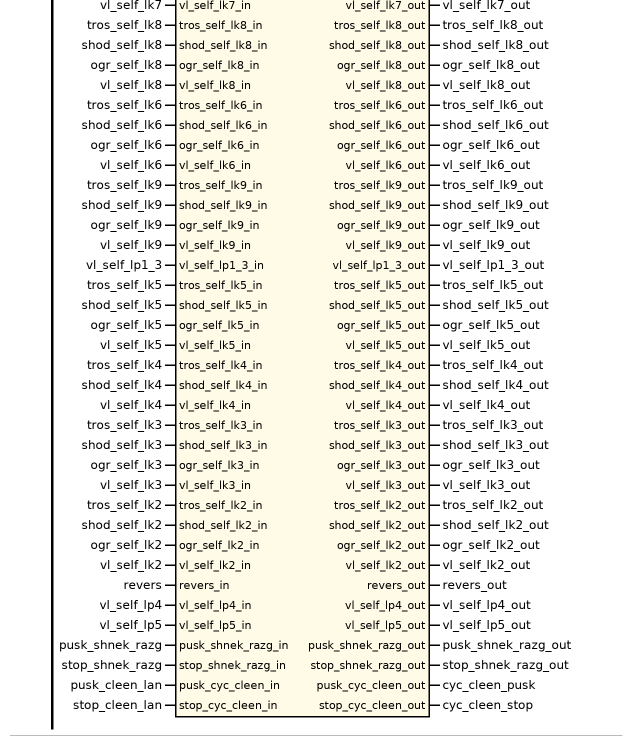
[picture p24: PLC_PRG (LD)]
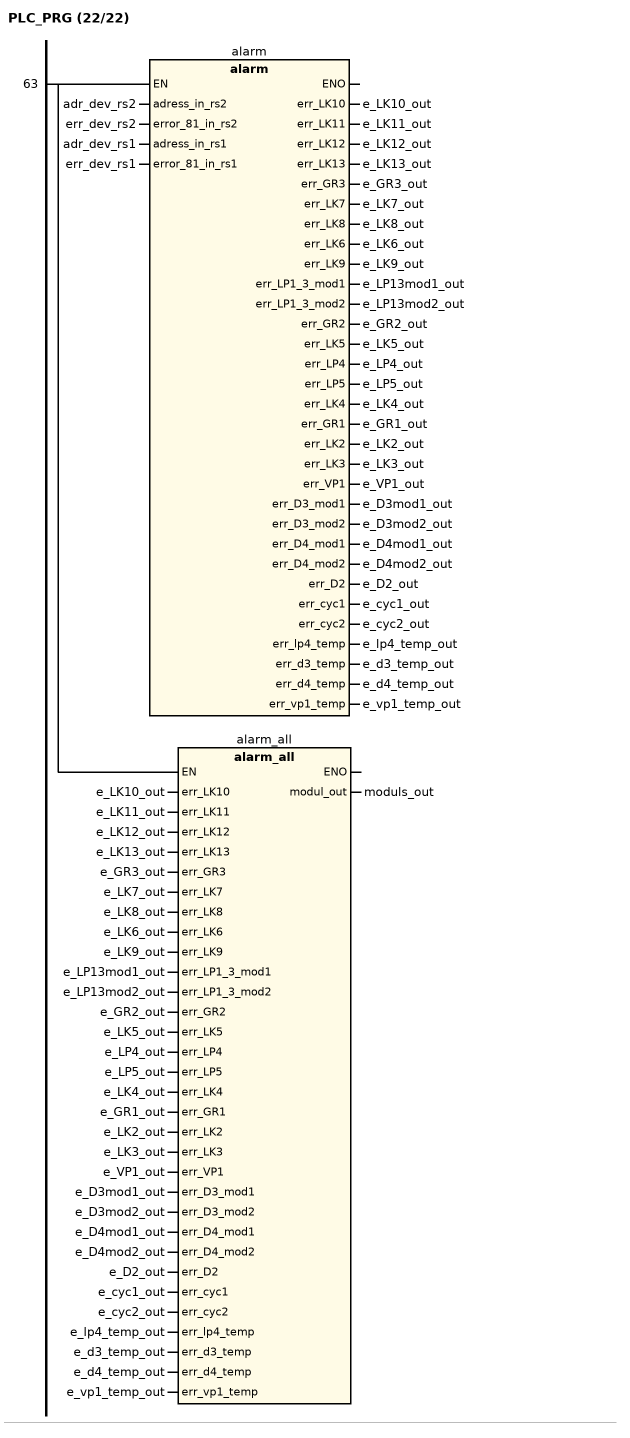
_LD_ (* Ladder Diagram *)
NETWORK 1 (* Фиксация пуска для SCADA-системы *)
	{ [pusk_sys] - [avto_all] | [pusk_lan] } - [/stop_DDD] - [/gribok] --- (pusk_lan)
NETWORK 2 (* Пуск только по готовностям всех шкафов *)
	[pusk_sys] - [avto_all] - [ready_D2] - [ready_D3] - { [ready_D4] | [in_040] } - [ready_LK10] - [ready_LK11] - { [ready_LK12] | [/current_value_lk_glob] } - [ready_LK13] - [ready_GR3] - { [ready_LK7] | [in_040] } - [ready_LK8] - [ready_LK9] - { [ready_LK6] | [in_020] } - [ready_LP1_3] - [ready_GR2] - [ready_LK5] - [ready_LP4] - { [ready_LP5] | [in_040] } - [ready_GR1] - [ready_LK2] - [ready_VP1] - [ready_LK3] --- (pusk)
NETWORK 3 (* Остановка всех агрегатов по втором нажатии кнопки "стоп" *)
	[stop_sys] - stop:CTU(CU: *, RESET: stop_DDD OR pusk_sys OR ruchnoe_all, PV: 2) --- (stop_all)
NETWORK 4 (* Остановка дробилок по третьему нажатию кнопки "стоп" *)
	[stop_sys] - stop_Drob:CTU(CU: *, RESET: stop_DDD OR pusk_sys, PV: 3) --- (stop_D2)
NETWORK 5
	*
		EN --- cyclone:cyclone(stop: stop_DDD, grib: gribok, pusk_LAN: pusk_lan_cyclone_out, stop_lan: stop_lan_cyclone_out, level: lev_up_cyc, KU: ku_cyc, TZ: tz_cyc, skvaj: skvaj_in, switch: revers_out, err: e_cyc1_out OR e_cyc2_out, pusk_shnek_lan: pusk_shnek_razg_out, stop_shnek_lan: stop_shnek_razg_out, in_time: in_time_shake, time_run: time_run, time_stop: time_stop, cleen_in_pusk: cyc_cleen_pusk, cleen_in_stop: cyc_cleen_stop, VE_1 => ve1_out, VE_2 => ve2_out, VE_3 => ve3_out, VE_4 => ve4_out, VE_5 => ve5_out, VE_6 => ve6_out, VE_7 => ve7_out, VE_8 => ve8_out, shnek_up => shnek_up_cyc, ready => ready_cyc, work => work_cyc, avar => avar_cyc, shnek_razg => shnek_razg, prom_cleen_word => prom_cleen_out) => vent_pump_cyc
NETWORK 6
	*
		EN --- PACK(shnek_razg, vent_pump_cyc, shnek_up_cyc, FALSE, FALSE, FALSE, FALSE, FALSE) => km_byte_cyc
NETWORK 7 (* Блок управления дробилкой Д2 *)
	[pusk] - D2:D2(pusk: *, KUD2: KU_D2, RMS2_2: RMS2_2, RD2: RD2_D2, TZD2: TZD2, avto: avto_D2, GRIB: gribok, stop_s: stop_D2, ruchnoe: ruchnoe_all, pusk_LAN: pusk_LAN_D2_out, stop_LAN: stop_LAN_D2_out, err: e_D2_out, work => work_D2, KM2 => KM2_D2, KM3 => KM3_D2, stop_D3D4 => stop_D3, avar => avar_D2) --- (ready_D2)
NETWORK 8 (* Блок управления битовой маской выходов модуля расширения в шкафу управления Д2 *)
	*
		EN --- PACK(FALSE, KM2_D2, FALSE, KM3_D2, FALSE, FALSE, FALSE, FALSE) => KM_D2_byte
NETWORK 9 (* Блок управления дробилкой Д3 *)
	[pusk] - D3:D3(pusk: *, KU: KU_D3, TZN: TZN_D3, KPM: KPM_D3, TZV: TZV_D3, KUD3: KUD3_D3, TZD3: TZD3_D3, RD3: RD3_D3, TM: TM_D3, RMS: RMS_D3, avto_in: avto_D3, GRIB: gribok, work_D2_D3: work_D2, stop_in: stop_D2, ruchnoe: ruchnoe_all, pusk_LAN: pusk_LAN_D3_out, stop_LAN: stop_LAN_D3_out, err: e_D3mod1_out OR e_D3mod2_out, UM: UM_D3, KM2 => KM2_D3, KM3 => KM3_D3, ready => ready_D3, nasos => nasos_D3, vent => vent_D3, ten => ten_D3, work => work_D3, avto => out_avto_D3, avar => avar_D3, stop_D3D4 => stop_D4, tm_ins => TM_D3_bool) --- (KM1_D3)
NETWORK 10 (* Блок управления битовой маской выходов модуля расширения в шкафу управления Д4 *)
	*
		EN --- PACK(out_avto_D3, nasos_D3, vent_D3, ten_D3, FALSE, FALSE, FALSE, FALSE) => D3_mod1_byte
		EN --- PACK(FALSE, KM1_D3, KM2_D3, KM3_D3, FALSE, FALSE, FALSE, FALSE) => D3_mod2_byte
NETWORK 11 (* Блок управления дробилкой Д4 *)
	[pusk] - D4:D4(pusk: *, KU: KU_D4, TZN: TZN_D4, KPM: KPM_D4, TZV: TZV_D4, KUD3: KUD3_D4, TZD3: TZD3_D4, RD3: RD3_D4, TM: TM_D4, RMS: RMS_D4, avto_in: avto_D4, GRIB: gribok, work_D2_D3: work_D3, stop_in: stop_D4, ruchnoe: ruchnoe_all, ins_0_40: in_040, pusk_LAN: pusk_LAN_D4_out, stop_LAN: stop_LAN_D4_out, err: e_D4mod1_out OR e_D4mod2_out, UM: UM_D4, KM2 => KM2_D4, KM3 => KM3_D4, ready => ready_D4, nasos => nasos_D4, vent => vent_D4, ten => ten_D4, work => work_D4, avto => out_avto_D4, avar => avar_D4, stop_D3D4 => stop_DDD, tm_ins => TM_D4_bool) --- (KM1_D4)
NETWORK 12 (* Блок управления битовой маской выходов модуля расширения в шкафу управления Д4 *)
	*
		EN --- PACK(out_avto_D4, nasos_D4, vent_D4, ten_D4, FALSE, FALSE, FALSE, FALSE) => D4_mod1_byte
		EN --- PACK(FALSE, KM1_D4, KM2_D4, KM3_D4, FALSE, FALSE, FALSE, FALSE) => D4_mod2_byte
NETWORK 13 (* Подтверждение работы дробилок Д2-Д4 и разрешение на пуск следующей ступени агрегатов *)
	[work_D2] - [work_D3] - { [work_D4] | [in_040] } --- (work_level_10)
NETWORK 14 (* Проверка готовностей ленточных конвееров ЛК10-ЛК13. После пуска всех агрегатов этой ступени, / промежуточное реле самоподхвата разрывается для защиты от повторного пуска *)
	{ [pusk] - [ready_LK10] - [ready_LK11] - [ready_LK13] | [prom1] - [/work_level_1] - [/avar_LK10] - [/avar_LK11] - [/avar_LK13] } - [/STOP_SYS] - [/stop_lan_LK10_out] - [/stop_lan_LK11_out] - [/stop_lan_LK13_out] --- (prom1)
NETWORK 15 (* Блок управления ленточным конвеером ЛК-10 *)
	[work_level_10] - ton_LK10:TON(IN: *, PT: t#1s) - [avto_all] - [prom1] - LK10:LK1(pusk: *, avto: avto_LK10, KU: KU_LK10, TZ: TZ_LK10, tros: tros_LK10, shod: shod_LK10, ogr: ogr_LK10, VL: bool_Vl_LK10, P: P_LK10, GRIB: gribok, stop_s: stop_all, ruchnoe: ruchnoe_all, pusk_LAN: pusk_lan_LK10_out, stop_LAN: stop_lan_LK10_out, err: e_LK10_out, tros_self: tros_self_lk10_out, shod_self: shod_self_lk10_out, ogr_self: ogr_self_lk10_out, pusk_sys_ins: PUSK_SYS, ready => ready_LK10, work => work_LK10, avar => avar_LK10, avar_vl => avar_vl_lk10) --- (KM1_LK10)
NETWORK 16 (* Блок управления ленточным конвеером ЛК-11 *)
	[work_LK10] - ton_lk11:TON(IN: *, PT: t#1s) - [avto_all] - [prom1] - LK11:LK1(pusk: *, avto: avto_LK11, KU: KU_LK11, TZ: TZ_LK11, tros: tros_LK11, shod: shod_LK11, ogr: ogr_LK11, VL: bool_Vl_LK11, P: P_LK11, GRIB: gribok, stop_s: stop_all, ruchnoe: ruchnoe_all, pusk_LAN: pusk_lan_LK11_out, stop_LAN: stop_lan_LK11_out, err: e_LK11_out, tros_self: tros_self_lk11_out, shod_self: shod_self_lk11_out, ogr_self: ogr_self_lk11_out, pusk_sys_ins: PUSK_SYS, ready => ready_LK11, work => work_LK11, avar => avar_LK11, avar_vl => avar_vl_lk11) --- (KM1_LK11)
NETWORK 17 (* Блок управления ленточным конвеером ЛК-12 *)
	[work_LK11] - ton_lk12:TON(IN: *, PT: t#1s) - [avto_all] - [prom1] - LK12:LK12_modern(pusk: *, avto: avto_LK12, KU: KU_LK12, TZ: TZ_LK12, tros: tros_LK12, shod: shod_LK12, ogr: ogr_LK12, VL: bool_Vl_LK12, P: P_LK12, GRIB: gribok, stop_s: stop_all, ruchnoe: ruchnoe_all, pusk_LAN: pusk_lan_LK12_out, stop_LAN: stop_lan_LK12_out, err: e_LK12_out, tros_self: tros_self_lk12_out, shod_self: shod_self_lk12_out, ogr_self: ogr_self_lk12_out, pusk_sys_ins: PUSK_SYS, switcher_in: lk12_switcher, current_value_lk12_in: current_value_lk_glob, ready => ready_LK12, work => work_LK12, avar => avar_LK12, avar_vl => avar_vl_lk12, current_value_lk12_out => current_value_lk_glob) --- (KM1_LK12)
NETWORK 18 (* Блок управления ленточным конвеером ЛК-13 *)
	[work_LK11] - ton_lk13:TON(IN: *, PT: t#1s) - [avto_all] - [prom1] - LK13:LK1(pusk: *, avto: avto_LK13, KU: KU_LK13, TZ: TZ_LK13, tros: tros_LK13, shod: shod_LK13, ogr: ogr_LK13, VL: bool_Vl_LK13, P: P_LK13, GRIB: gribok, stop_s: stop_all, ruchnoe: ruchnoe_all, pusk_LAN: pusk_lan_LK13_out, stop_LAN: stop_lan_LK13_out, err: e_LK13_out, tros_self: tros_self_lk13_out, shod_self: shod_self_lk13_out, ogr_self: ogr_self_lk13_out, pusk_sys_ins: PUSK_SYS, ready => ready_LK13, work => work_LK13, avar => avar_LK13, avar_vl => avar_vl_lk13) --- (KM1_LK13)
NETWORK 19 (* Подтверждение работы конвееров ЛК10-ЛК13 и разрешение на пуск следующей ступени агрегатов *)
	[work_LK10] - [work_LK11] - [work_LK13] --- (work_level_1)
NETWORK 20 (* Определить, какой из конвееров первой ветки остановился *)
	{ [avar_vl_lk10] | [avar_vl_lk11] | [avar_vl_lk13] } --- (stop_vl_lv1)
NETWORK 21 (* Проверка готовности грохота ГР3. После пуска агрегата, / промежуточное реле самоподхвата разрывается для защиты от повторного пуска *)
	{ [pusk] - [ready_GR3] | [prom2] - [/work_GR3] - [/avar_GR3] } - [/STOP_SYS] - [/stop_lan_GR3_out] --- (prom2)
NETWORK 22 (* Блок управления грохотом ГР3 *)
	[work_level_1] - ton_GR3:TON(IN: *, PT: t#1s) - [avto_all] - [prom2] - GR3:Grohot(pusk: *, avto: avto_GR3, KU: KU_gr3, TZ: TZ_gr3, P: p_gr3, STOP: STOP_GR3, GRIB: gribok, stop_s: stop_all, ruchnoe: ruchnoe_all, pusk_LAN: pusk_lan_GR3_out, stop_LAN: stop_lan_GR3_out, err: e_GR3_out, ready => ready_GR3, work => work_GR3, avar => avar_GR3) --- (KM1_GR3)
NETWORK 23 (* Подтверждение работы ступени №1 и грохота, и разрешение на пуск следующей ступени агрегатов *)
	[work_level_1] - [work_GR3] --- (work_level_2)
NETWORK 24 (* Проверка готовностей ленточных конвееров ЛК6,ЛК7-ЛК9. После пуска всех агрегатов этой ступени, / промежуточное реле самоподхвата разрывается для защиты от повторного пуска *)
	{ [pusk] - { [ready_LK7] | [in_040] } - [ready_LK8] - [ready_LK9] - { [ready_LK6] | [in_020] } | [prom3] - [/work_level_3] - [/avar_LK7] - [/avar_LK8] - [/avar_LK6] - [/avar_LK9] } - [/STOP_SYS] - [/stop_lan_LK7_out] - [/stop_lan_LK8_out] - [/stop_lan_LK6_out] - [/stop_lan_LK9_out] --- (prom3)
NETWORK 25 (* Блок управления ленточным конвеером ЛК-7 *)
	[work_GR3] - ton_LK7:TON(IN: *, PT: t#10s) - [avto_all] - [prom3] - LK7:LK3(pusk: *, avto: avto_LK7, KU: KU_LK7, TZ: TZ_LK7, tros: tros_LK7, shod: shod_LK7, ogr: ogr_LK7, VL: bool_Vl_LK7, P: P_LK7, in_020: in_040, stop_s: stop_all, GRIB: gribok, ruchnoe: ruchnoe_all, pusk_LAN: pusk_lan_LK7_out, stop_LAN: stop_lan_LK7_out, err: e_LK7_out, tros_self: tros_self_lk7_out, shod_self: shod_self_lk7_out, ogr_self: ogr_self_lk7_out, pusk_sys_ins: PUSK_SYS, ready => ready_LK7, work => work_LK7, avar => avar_LK7, avar_vl => avar_vl_lk7) --- (KM1_LK7)
NETWORK 26 (* Блок управления ленточным конвеером ЛК-8 *)
	{ [work_LK7] - ton_LK8:TON(IN: *, PT: t#1s) | [work_GR3] - [in_040] - ton_LK81:TON(IN: *, PT: t#10s) } - [avto_all] - [prom3] - LK8:LK1(pusk: *, avto: avto_LK8, KU: KU_LK8, TZ: TZ_LK8, tros: tros_LK8, shod: shod_LK8, ogr: ogr_LK8, VL: bool_Vl_LK8, P: P_LK8, GRIB: stop_all, stop_s: gribok, ruchnoe: ruchnoe_all, pusk_LAN: pusk_lan_LK8_out, stop_LAN: stop_lan_LK8_out, err: e_LK8_out, tros_self: tros_self_lk8_out, shod_self: shod_self_lk8_out, ogr_self: ogr_self_lk8_out, pusk_sys_ins: PUSK_SYS, ready => ready_LK8, work => work_LK8, avar => avar_LK8, avar_vl => avar_vl_lk8) --- (KM1_LK8)
NETWORK 27 (* Блок управления ленточным конвеером ЛК-6 *)
	[work_LK8] - ton_LK6:TON(IN: *, PT: t#1s) - [avto_all] - [prom3] - LK6:LK3(pusk: *, avto: avto_LK6, KU: KU_LK6, TZ: TZ_LK6, tros: tros_LK6, shod: shod_LK6, ogr: ogr_LK6, VL: bool_Vl_LK6, P: P_LK6, in_020: in_020, stop_s: stop_all, GRIB: gribok, ruchnoe: ruchnoe_all, pusk_LAN: pusk_lan_LK6_out, stop_LAN: stop_lan_LK6_out, err: e_LK6_out, tros_self: tros_self_lk6_out, shod_self: shod_self_lk6_out, ogr_self: ogr_self_lk6_out, pusk_sys_ins: PUSK_SYS, ready => ready_LK6, work => work_LK6, avar => avar_LK6, avar_vl => avar_vl_lk6) --- (KM1_LK6)
NETWORK 28 (* Блок управления ленточным конвеером ЛК-9 *)
	{ [work_LK6] | [in_020] - [work_LK8] } - ton_LK9:TON(IN: *, PT: t#1s) - [avto_all] - [prom3] - LK9:LK1(pusk: *, avto: avto_LK9, KU: KU_LK9, TZ: TZ_LK9, tros: tros_LK9, shod: shod_LK9, ogr: ogr_LK9, VL: bool_Vl_LK9, P: P_LK9, GRIB: gribok, stop_s: stop_all, ruchnoe: ruchnoe_all, pusk_LAN: pusk_lan_LK9_out, stop_LAN: stop_lan_LK9_out, err: e_LK9_out, tros_self: tros_self_lk9_out, shod_self: shod_self_lk9_out, ogr_self: ogr_self_lk9_out, pusk_sys_ins: PUSK_SYS, ready => ready_LK9, work => work_LK9, avar => avar_LK9, avar_vl => avar_vl_lk9) --- (KM1_LK9)
NETWORK 29
	{ [avar_vl_lk7] | [avar_vl_lk8] | [avar_vl_lk6] | [avar_vl_lk9] | [stop_vl_lv1] } --- (stop_vl_lv2)
NETWORK 30 (* Подтверждение работы конвееров ЛК6,ЛК7-ЛК9 и разрешение на пуск следующей ступени агрегатов *)
	{ [work_LK7] | [in_040] } - [work_LK8] - { [work_LK6] | [in_020] } - [work_LK9] --- (work_level_3)
NETWORK 31 (* Проверка готовности ленточного питателя ЛП1-ЛП3. После пуска всех агрегатов этой ступени, / промежуточное реле самоподхвата разрывается для защиты от повторного пуска *)
	{ [pusk] - [ready_LP1_3] | [prom4] - [/work_LP1_3] - [/avar_LP1_3] } - [/STOP_SYS] - [/stop_lan_LP1_3_out] --- (prom4)
NETWORK 32 (* Блок управления ленточным питетелем ЛП1-ЛП3 *)
	[work_LK9] - ton_LP1_3:TON(IN: *, PT: t#1s) - [avto_all] - [prom4] - LP1_3:LP1_3(pusk_sys: *, Vl1: TRUE, Vl2: TRUE, Vl3: TRUE, in_020: in_020, in_040: in_040, in_020_4070: in_020_4070, KU: KU_LP1_3, TZ1: TZ1_LP1_3, TZ2: TZ2_LP1_3, TZ3: TZ3_LP1_3, PRO: PRO_LP1_3, avto: avto_LP1_3, P: P_LP1_3, stop2: stop2_LP1_3, GRIB: gribok, stop_s: stop_all, ruchnoe: ruchnoe_all, pusk_LAN: pusk_lan_LP1_3_out, stop_LAN: stop_lan_LP1_3_out, err: e_LP13mod1_out OR e_LP13mod2_out, pusk_sys_ins: PUSK_SYS, KM2 => KM2_LP1_3, KM4 => KM4_LP1_3, KM5 => KM5_LP1_3, KM3 => KM3_LP1_3, ready => ready_LP1_3, work => work_LP1_3, avar => avar_LP1_3, avar_vl => avar_vl_lp1_3) --- (KM1_LP1_3)
NETWORK 33 (* Блок управления битовой маской выходов модуля расширения в шкафу управления ЛП1-ЛП3 *)
	*
		EN --- PACK(KM2_LP1_3, KM3_LP1_3, KM4_LP1_3, KM5_LP1_3, FALSE, FALSE, FALSE, FALSE) => KM2345_LP1_3_byte
NETWORK 34 (* Проверка готовности грохота ГР2. После пуска всех агрегатов этой ступени, / промежуточное реле самоподхвата разрывается для защиты от повторного пуска *)
	{ [pusk] - [ready_GR2] | [prom5] - [/avar_GR2] - [/work_GR2] } - [/STOP_SYS] - [/stop_lan_GR2_out] --- (prom5)
NETWORK 35 (* Блок управления грохотом ГР2 *)
	[work_LP1_3] - ton_GR2:TON(IN: *, PT: t#1s) - [avto_all] - [prom5] - GR2:Grohot1(pusk: *, avto: avto_GR2, KU: KU_GR2, TZ: TZ_GR2, P: P_GR2, STOP: STOP_GR2, stop_sys: gribok, GRIB: stop_all, stop_lv: work_LP1_3, ruchnoe: ruchnoe_all, pusk_LAN: pusk_lan_GR2_out, stop_LAN: stop_lan_GR2_out, err: e_GR2_out, ready => ready_GR2, work => work_GR2, avar => avar_GR2) --- (KM1_GR2)
NETWORK 36 (* Подтверждение работы ГР2, ЛП1-ЛП3 и разрешение на пуск следующей ступени агрегатов *)
	[work_level_3] - [work_GR2] --- (work_level_4)
NETWORK 37
	{ [avar_vl_lk7] | [avar_vl_lk8] | [avar_vl_lk6] | [avar_vl_lk9] | [avar_vl_lp1_3] | [stop_vl_lv1] } --- (stop_vl_lv2)
NETWORK 38 (* Проверка готовности ленточного конвеера ЛК5. После пуска всех агрегатов этой ступени, / промежуточное реле самоподхвата разрывается для защиты от повторного пуска *)
	{ [pusk] - [ready_LK5] | [prom6] - [/avar_LK5] - [/work_LK5] } - [/STOP_SYS] - [/stop_lan_LK5_out] --- (prom6)
NETWORK 39 (* Блок управления ленточного конвеера ЛК5 *)
	[work_GR2] - ton_LK5:TON(IN: *, PT: t#10s) - [avto_all] - [prom6] - LK5:LK1(pusk: *, avto: avto_LK5, KU: KU_LK5, TZ: TZ_LK5, tros: tros_LK5, shod: shod_LK5, ogr: ogr_LK5, VL: bool_Vl_LK5, P: P_LK5, GRIB: gribok, stop_s: stop_all, ruchnoe: ruchnoe_all, pusk_LAN: pusk_lan_LK5_out, stop_LAN: stop_lan_LK5_out, err: e_LK5_out, tros_self: tros_self_lk5_out, shod_self: shod_self_lk5_out, ogr_self: ogr_self_lk5_out, pusk_sys_ins: PUSK_SYS, ready => ready_LK5, work => work_LK5, avar => avar_LK5, avar_vl => avar_vl_lk5) --- (KM1_LK5)
NETWORK 40 (* Подтверждение работы дробилки Д3 и ленточного конвеера ЛК5, и разрешение на пуск следующей ступени агрегатов *)
	[work_D3] - [work_LK5] - [work_level_2] - [work_level_4] --- (work_level_6)
NETWORK 41 (* Подтверждение работы дробилки Д4, ленточного конвеера ЛК5, "куста" №1, "куста" №2 и разрешение на пуск следующей ступени агрегатов *)
	[work_D4] - [work_LK5] - [work_level_2] - [work_level_4] --- (work_level_61)
NETWORK 42 (* Проверка готовности ленточных питателей ЛП4 и ЛП5. После пуска всех агрегатов этой ступени, / промежуточное реле самоподхвата разрывается для защиты от повторного пуска *)
	{ [pusk] - [ready_LP4] - { [ready_LP5] | [in_040] } | [prom7] - [/work_LP4] - [/work_LP5] } - [/STOP_SYS] - [/stop_LAN_LP4_out] - [/stop_LAN_LP5_out] --- (prom7)
NETWORK 43 (* Блок управления ленточного питателя ЛП4 *)
	[work_LK5] - [avto_all] - [prom7] - LP4:LP4_without_FC(pusk: *, avto: avto_LP4, KU: KU_LP4, TZ: TZ_LP4, MD3: MD2_LP4, P: P_LP4, stop_lv: work_level_6, GRIB: gribok, stop_s: stop_all, ruchnoe: ruchnoe_all, pusk_LAN: pusk_LAN_LP4_out, stop_LAN: stop_LAN_LP4_out, err: e_LP4_out, ready => ready_LP4, work => work_LP4, avar => avar_LP4, metall_LK4 => metall_LP4) --- (KM1_LP4)
NETWORK 44 (* Блок управления ленточного питателя ЛП5 *)
	[work_LK5] - [avto_all] - [prom7] - LP5:LP5(pusk: *, avto: avto_LP5, STOP: STOP_LP5, VL: TRUE, MD2: MD2_LP5, stop_lv: work_level_61, GRIB: gribok, input_Hz: out_Hz_LP5, stop_s: stop_all, pusk_LAN: pusk_LAN_LP5_out, stop_LAN: stop_LAN_LP5_out, P: in_P_LP5, ruchnoe: ruchnoe_all, ins_0_40: in_040, err: e_LP5_out, pusk_sys_ins: PUSK_SYS, avar_FC: avar_FC_LP5, KM => pusk_LP5, work => work_LP5, avar => avar_LP5, met => metall_LP5, b1_00 => b1_00_LP5, b1_04 => b1_04_LP5, avto_in => avto_out_LP5, avar_vl => avar_vl_lp5) --- (ready_LP5)
NETWORK 45
	{ [avar_vl_lk5] | [stop_vl_lv2] } --- (stop_vl_lv3)
NETWORK 46 (* Проверка готовности ленточного конвеера ЛК4. После пуска всех агрегатов этой ступени, / промежуточное реле самоподхвата разрывается для защиты от повторного пуска *)
	{ [pusk] - [ready_LK4] | [prom8] - [/avar_LK4] - [/work_LK4] } - [/STOP_SYS] - [/stop_lan_LK4_out] --- (prom8)
NETWORK 47 (* Блок управления ленточного конвеера ЛК4 *)
	[work_LK5] - ton_LK4:TON(IN: *, PT: t#1s) - [avto_all] - [prom8] - LK4:LK4(pusk: *, avto: avto_LK4, KU: KU_LK4, TZ: TZ_LK4, tros: tros_LK4, shod: shod_LK4, MD3: MD3_LK4, VL: bool_Vl_LK4, P: P_LK4, stop_lv: work_D2 AND work_level_4 AND work_lk5 AND work_level_2, GRIB: gribok, stop_s: stop_all, ruchnoe: ruchnoe_all, pusk_LAN: pusk_lan_LK4_out, stop_LAN: stop_lan_LK4_out, err: e_LK4_out, tros_self: tros_self_lk4_out, shod_self: shod_self_lk4_out, pusk_sys_ins: PUSK_SYS, ready => ready_LK4, work => work_LK4, avar => avar_LK4, metall_LK4 => metall_LK4, avar_vl => avar_vl_lk4) --- (KM1_LK4)
NETWORK 48
	{ [pusk] - [ready_VP1] | [prom10] - [/work_VP1] - [/avar_VP1] } - [/STOP_SYS] - [/stop_LAN_VP1_out] --- (prom10)
NETWORK 49 (* Блок управления вибропитателя ВП1 *)
	[work_LK4] - [avto_all] - [prom10] - VP1:VP1(pusk: *, avto: avto_VP1, KU: KU_VP1, TZ: TZ_VP1, STOP: STOP_VP1, stop_lv: work_LK4, GRIB: gribok, LV_low_LK7: TRUE, LV_high_LK7: FALSE, LV_low_LK8: TRUE, LV_high_LK8: FALSE, LV_low_D2: LV_low_D2, LV_high_D2: LV_high_D2, stop_s: stop_all, pusk_LAN: pusk_LAN_VP1_out, stop_LAN: stop_LAN_VP1_out, P: P_VP1, err: e_VP1_out OR e_lp4_temp_out, KM => pusk_VP1, work => work_VP1, avar => avar_VP1) --- (ready_VP1)
NETWORK 50 (* Проверка готовности ленточного конвеера ЛК2, ЛК3, грохота ГР1 и вибропитателя ВП1. После пуска всех агрегатов этой ступени, / промежуточное реле самоподхвата разрывается для защиты от повторного пуска *)
	{ [pusk] - [ready_GR1] - [ready_LK2] - [ready_LK3] | [prom9] - [/work_level_9] - [/avar_LK3] - [/avar_LK2] - [/avar_VP1] } - [/STOP_SYS] - [/stop_lan_LK3_out] - [/stop_lan_GR1_out] - [/stop_lan_LK2_out] --- (prom9)
NETWORK 51 (* Блок управления ленточного конвеера ЛК3 *)
	[work_LK4] - ton_LK3:TON(IN: *, PT: t#1s) - [avto_all] - [prom9] - LK3:LK1(pusk: *, avto: avto_LK3, KU: KU_LK3, TZ: TZ_LK3, tros: tros_LK3, shod: shod_LK3, ogr: ogr_LK3, VL: bool_Vl_LK3, P: P_LK3, GRIB: stop_all, stop_s: gribok, ruchnoe: ruchnoe_all, pusk_LAN: pusk_lan_LK3_out, stop_LAN: stop_lan_LK3_out, err: e_LK3_out, tros_self: tros_self_lk3_out, shod_self: shod_self_lk3_out, ogr_self: ogr_self_lk3_out, pusk_sys_ins: PUSK_SYS, ready => ready_LK3, work => work_LK3, avar => avar_LK3, avar_vl => avar_vl_lk3) --- (KM1_LK3)
NETWORK 52 (* Блок управления грохота ГР1 *)
	[work_LK3] - ton_GR1:TON(IN: *, PT: t#1s) - [avto_all] - [prom9] - GR1:Grohot(pusk: *, avto: avto_GR1, KU: KU_GR1, TZ: TZ_GR1, P: P_GR1, STOP: STOP_GR1, GRIB: stop_all, stop_s: gribok, ruchnoe: ruchnoe_all, pusk_LAN: pusk_lan_GR1_out, stop_LAN: stop_lan_GR1_out, err: e_GR1_out, ready => ready_GR1, work => work_GR1, avar => avar_GR1) --- (KM1_GR1)
NETWORK 53 (* Блок управления ленточного конвеера ЛК2 *)
	[work_GR1] - ton_LK2:TON(IN: *, PT: t#10s) - [avto_all] - [prom9] - LK2:LK2(pusk: *, avto: avto_LK2, KU: KU_LK2, TZ: TZ_LK2, tros: tros_LK2, shod: shod_LK2, ogr: ogr_LK2, VL: bool_Vl_LK2, P: P_LK2, GRIB: gribok, stop_s: stop_all, stop_lv: work_GR1, ruchnoe: ruchnoe_all, pusk_LAN: pusk_lan_LK2_out, stop_LAN: stop_lan_LK2_out, err: e_LK2_out, tros_self: tros_self_lk2_out, shod_self: shod_self_lk2_out, ogr_self: ogr_self_lk2_out, pusk_sys_ins: PUSK_SYS, ready => ready_LK2, work => work_LK2, avar => avar_LK2, avar_vl => avar_vl_lk2) --- (KM1_LK2)
NETWORK 54 (* Подтверждение работы ленточных конвееров ЛК2, ЛК3, грохота ГР1 и вибропитателя ВП1 *)
	[work_LK2] - [work_LK3] - [work_GR1] --- (work_level_9)
NETWORK 55 (* Блок отключения пластинчатого питателя ПП1 *)
	*
		EN --- PP1_blok:PP1(P_LK2_in: work_LK2, stop_pp_LK3: work_LK3, LV2: LV_low_GR1, LV1: LV_high_GR1, pusk_s: pusk_sys, stop_s: stop_sys) => PP1
NETWORK 56 (* Блок управления битовой маской выходов модуля расширения в шкафу управления ЛК2 *)
	*
		EN --- PACK(KM1_LK2, FALSE, PP1, FALSE, FALSE, FALSE, FALSE, FALSE) => LK2_out
NETWORK 57 (* Блоки управления отключением вибропитателя ВП1, ленточных конвееров ЛК7 и ЛК8 в зависимости от уровня в бункере *)
	*
		EN --- stop_VP1_LK7:stop_VP1(LV_in: 4-LV_LK7, LV_high_in: ust_LV2_LK7, LV_low_in: ust_LV1_LK7, LV1_out => LV_low_LK7) => LV_high_LK7
		EN --- stop_VP1_LK8:stop_VP1(LV_in: 4-LV_LK8, LV_high_in: ust_LV2_LK8, LV_low_in: ust_LV1_LK8, LV1_out => LV_low_LK8) => LV_high_LK8
		EN --- stop_VP1_D2:stop_VP1(LV_in: 2.2-LV_D2, LV_high_in: ust_LV2_D2, LV_low_in: ust_LV1_D2, LV1_out => LV_low_D2) => LV_high_D2
		EN --- stop_PP1:stop_VP1(LV_in: LV_GR1 - 0.8, LV_high_in: ust_LV2_GR1, LV_low_in: ust_LV1_GR1, LV1_out => LV_low_GR1) => LV_high_GR1
		EN --- if_Hz:if_Hz(input_Hz_LP4_if: input_Hz_LP4, input_Hz_LP5_if: input_Hz_LP5, output_Hz_LP5_if => out_Hz_LP5) => out_Hz_LP4
		EN --- if_LV:if_LV(input_LV2_LK7: ust_LV2_LK7, input_LV1_LK7: ust_LV1_LK7, input_LV2_LK8: ust_LV2_LK8, input_LV1_LK8: ust_LV1_LK8, input_LV2_GR1: ust_LV2_GR1, input_LV1_GR1: ust_LV1_GR1, input_LV2_D2: ust_LV2_D2, input_LV1_D2: ust_LV1_D2, input_time_VL: time_VL, output_LV1_LK7 => ust_LV1_LK7, output_LV2_LK8 => ust_LV2_LK8, output_LV1_LK8 => ust_LV1_LK8, output_LV2_GR1 => ust_LV2_GR1, output_LV1_GR1 => ust_LV1_GR1, output_LV2_D2 => ust_LV2_D2, output_LV1_D2 => ust_LV1_D2, output_time_VL => time_VL) => ust_LV2_LK7
NETWORK 58 (* Вывод аварии, в виде световой сигнализации, на шкаф контроллера *)
	{ [avar_D3] | [avar_D4] | [avar_LK10] | [avar_LK11] | [avar_LK12] | [avar_LK13] | [avar_GR3] | [avar_LK7] | [avar_LK6] | [avar_LK9] | [avar_LP1_3] | [avar_GR2] | [avar_LK5] | [avar_LP4] | [avar_LP5] | [avar_GR1] | [avar_LK4] | [avar_Lk2] | [avar_VP1] | [avar_LK3] | [gribok] } --- (avaria)
NETWORK 59 (* Вывод наличия, в виде световой сигнализации, на шкаф контроллера *)
	{ [metall_LP4] | [metall_LP5] | [metall_LK4] } --- (metall)
NETWORK 60 (* Блоки управления подсчетом скорости вращения *)
	*
		EN --- counter_LK10:counter(Vl: Vl_LK10, work: work_lk10, in_time: time_VL) => bool_Vl_LK10
		EN --- counter_LK11:counter(Vl: Vl_LK11, work: work_lk11, in_time: time_VL) => bool_Vl_LK11
		EN --- counter_LK12:counter(Vl: Vl_LK12, work: work_lk12, in_time: time_VL) => bool_Vl_LK12
		EN --- counter_LK13:counter(Vl: Vl_LK13, work: work_lk13, in_time: time_VL) => bool_Vl_LK13
		EN --- counter_LK7:counter_lk5(Vl: Vl_LK7, work: work_lk7, in_time: time_VL) => bool_Vl_LK7
		EN --- counter_LK8:counter_lk5(Vl: Vl_LK8, work: work_lk8, in_time: time_VL) => bool_Vl_LK8
		EN --- counter_LK6:counter(Vl: Vl_LK6, work: work_lk6, in_time: time_VL) => bool_Vl_LK6
		EN --- counter_LK9:counter(Vl: Vl_LK9, work: work_lk9, in_time: time_VL) => bool_Vl_LK9
		EN --- counter_LP1_3_1:counter(Vl: Vl1_LP1_3, work: work_LP1_3, in_time: time_VL) => bool_Vl1_LP1_3
		EN --- counter_LP1_3_2:counter(Vl: Vl2_LP1_3, work: work_LP1_3, in_time: time_VL) => bool_Vl2_LP1_3
		EN --- counter_LP1_3_3:counter(Vl: Vl3_LP1_3, work: work_LP1_3, in_time: time_VL) => bool_Vl3_LP1_3
		EN --- counter_LK5:counter_lk5(Vl: Vl_LK5, work: work_lk5, in_time: time_VL) => bool_Vl_LK5
		EN --- counter_LP5:counter(Vl: Vl_LP5, work: work_lp5, in_time: time_VL) => bool_Vl_LP5
		EN --- counter_LK4:counter(Vl: Vl_LK4, work: work_lk4, in_time: time_VL) => bool_Vl_LK4
		EN --- counter_LK3:counter(Vl: Vl_LK3, work: work_lk3, in_time: time_VL) => bool_Vl_LK3
		EN --- counter_LK2:counter(Vl: Vl_LK2, work: work_lk2, in_time: time_VL) => bool_Vl_LK2
NETWORK 61 (* Блок вывода сигналов для SCADA-системы *)
	*
		EN --- signals:signals(KU_D2_in: KU_D2, RMS2_2_in: RMS2_2, avto_D2_in: avto_D2, work_D2_in: work_D2, ready_D2_in: ready_D2, TZD2_in: TZD2, KU_D3_in: KU_D3, TZN_D3_in: TZN_D3, UM_D3_in: UM_D3, KPM_D3_in: KPM_D3, TZV_D3_in: TZV_D3, avto_D3_in: avto_D3, KUD3_D3_in: KUD3_D3, TZD3_D3_in: TZD3_D3, work_D3_in: work_D3, ready_D3_in: ready_D3, TM_D3_in: TM_D3_bool, RMS_D3_in: RMS_D3, DM_D3_in: DM_D3, KU_D4_in: KU_D4, TZN_D4_in: TZN_D4, UM_D4_in: UM_D4, KPM_D4_in: KPM_D4, TZV_D4_in: TZV_D4, avto_D4_in: avto_D4, KUD3_D4_in: KUD3_D4, TZD3_D4_in: TZD3_D4, work_D4_in: work_D4, ready_D4_in: ready_D4, TM_D4_in: TM_D4_bool, RMS_D4_in: RMS_D4, DM_D4_in: DM_D4, KU_LK10_in: KU_LK10, TZ_LK10_in: TZ_LK10, tros_LK10_in: tros_LK10, shod_LK10_in: shod_LK10, ogr_LK10_in: ogr_LK10, avto_LK10_in: avto_LK10, ready_LK10_in: ready_LK10, work_LK10_in: work_LK10, KU_LK11_in: KU_LK11, TZ_LK11_in: TZ_LK11, tros_LK11_in: tros_LK11, shod_LK11_in: shod_LK11, ogr_LK11_in: ogr_LK11, avto_LK11_in: avto_LK11, ready_LK11_in: ready_LK11, work_LK11_in: work_LK11, KU_LK12_in: KU_LK12, TZ_LK12_in: TZ_LK12, tros_LK12_in: tros_LK12, shod_LK12_in: shod_LK12, ogr_LK12_in: ogr_LK12, avto_LK12_in: avto_LK12, ready_LK12_in: ready_LK12, work_LK12_in: work_LK12, KU_LK13_in: KU_LK13, TZ_LK13_in: TZ_LK13, tros_LK13_in: tros_LK13, shod_LK13_in: shod_LK13, ogr_LK13_in: ogr_LK13, avto_LK13_in: avto_LK13, ready_LK13_in: ready_LK13, work_LK13_in: work_LK13, avto_GR3_in: avto_GR3, KU_GR3_in: KU_GR3, TZ_GR3_in: TZ_GR3, ready_GR3_in: ready_GR3, work_GR3_in: work_GR3, STOP_GR3_in: STOP_GR3, KU_LK7_in: KU_LK7, TZ_LK7_in: TZ_LK7, tros_LK7_in: tros_LK7, shod_LK7_in: shod_LK7, ogr_LK7_in: ogr_LK7, avto_LK7_in: avto_LK7, ready_LK7_in: ready_LK7, work_LK7_in: work_LK7, KU_LK8_in: KU_LK8, TZ_LK8_in: TZ_LK8, tros_LK8_in: tros_LK8, shod_LK8_in: shod_LK8, ogr_LK8_in: ogr_LK8, avto_LK8_in: avto_LK8, ready_LK8_in: ready_LK8, work_LK8_in: work_LK8, KU_LK6_in: KU_LK6, TZ_LK6_in: TZ_LK6, tros_LK6_in: tros_LK6, shod_LK6_in: shod_LK6, ogr_LK6_in: ogr_LK6, avto_LK6_in: avto_LK6, ready_LK6_in: ready_LK6, work_LK6_in: work_LK6, KU_LK9_in: KU_LK9, TZ_LK9_in: TZ_LK9, tros_LK9_in: tros_LK9, ogr_LK9_in: ogr_LK9, shod_LK9_in: shod_LK9, avto_LK9_in: avto_LK9, ready_LK9_in: ready_LK9, work_LK9_in: work_LK9, KU_LP1_3_in: KU_LP1_3, in_020_in: in_020, in_040_in: in_040, in_020_4070_in: in_020_4070, TZ1_LP1_3_in: TZ1_LP1_3, TZ2_LP1_3_in: TZ2_LP1_3, TZ3_LP1_3_in: TZ3_LP1_3, PRO_LP1_3_in: PRO_LP1_3, avto_LP1_3_in: avto_LP1_3, ready_LP1_3_in: ready_LP1_3, work_LP1_3_in: work_LP1_3, stop2_LP1_3_in: stop2_LP1_3, avto_GR2_in: avto_GR2, KU_GR2_in: KU_GR2, TZ_GR2_in: TZ_GR2, ready_GR2_in: ready_GR2, work_GR2_in: work_GR2, STOP_GR2_in: STOP_GR2, KU_LK5_in: KU_LK5, TZ_LK5_in: TZ_LK5, tros_LK5_in: tros_LK5, shod_LK5_in: shod_LK5, ogr_LK5_in: ogr_LK5, avto_LK5_in: avto_LK5, ready_LK5_in: ready_LK5, work_LK5_in: work_LK5, KU_LK4_in: KU_LK4, TZ_LK4_in: TZ_LK4, tros_LK4_in: tros_LK4, shod_LK4_in: shod_LK4, avto_LK4_in: avto_LK4, ready_LK4_in: ready_LK4, work_LK4_in: work_LK4, MD3_LK4_in: metall_LK4, avto_GR1_in: avto_GR1, KU_GR1_in: KU_GR1, TZ_GR1_in: TZ_GR1, ready_GR1_in: ready_GR1, work_GR1_in: work_GR1, STOP_GR1_in: STOP_GR1, KU_LK2_in: KU_LK2, TZ_LK2_in: TZ_LK2, tros_LK2_in: tros_LK2, shod_LK2_in: shod_LK2, ogr_LK2_in: ogr_LK2, avto_LK2_in: avto_LK2, ready_LK2_in: ready_LK2, work_LK2_in: work_LK2, KU_LK3_in: KU_LK3, TZ_LK3_in: TZ_LK3, tros_LK3_in: tros_LK3, shod_LK3_in: shod_LK3, ogr_LK3_in: ogr_LK3, avto_LK3_in: avto_LK3, ready_LK3_in: ready_LK3, work_LK3_in: work_LK3, avto_LP4_in: avto_LP4, ready_LP4_in: ready_LP4, work_LP4_in: work_LP4, MD2_LP4_in: metall_LP4, avto_LP5_in: avto_LP5, ready_LP5_in: ready_LP5, work_LP5_in: work_LP5, STOP_LP5_in: STOP_LP5, output_Hz_LP5_in: output_Hz_LP5, MD2_LP5_in: metall_LP5, avto_VP1_in: avto_VP1, ready_VP1_in: ready_VP1, work_VP1_in: work_VP1, STOP_VP1_in: STOP_VP1, KU_VP1_in: KU_VP1, TZ_VP1_in: TZ_VP1, avto_all_in: avto_all, pusk_in: pusk_lan, PP1_in: PP1, LV_GR1_in: LV_GR1, LV_LK7_in: LV_LK7, LV_LK8_in: LV_LK8, LV_D2_in: LV_D2, lev_up_cyc_in: lev_up_cyc, pre_cyc_in: pre_cyc, ku_cyc_in: ku_cyc, tz_cyc_in: tz_cyc, ready_cyc_in: ready_cyc, work_cyc_in: work_cyc, shnek_up_cyc_in: shnek_up_cyc, avar_cyc_in: avar_cyc, gribok_in: gribok, TM_D3_word_in: TM_D3, TM_D4_word_in: TM_D4, avar_FC_lp5_in: avar_FC_LP5, lev_down_cyc_in: lev_down_cyc, RMS2_2_out => RMS_2_2_out, avto_D2_out => avto_D2_out, work_D2_out => work_D2_out, ready_D2_out => ready_D2_out, TZD2_out => TZD2_out, KU_D3_out => KU_D3_out, TZN_D3_out => TZN_D3_out, UM_D3_out => UM_D3_out, KPM_D3_out => KPM_D3_out, TZV_D3_out => TZV_D3_out, avto_D3_out => avto_D3_out, KUD3_D3_out => KUD3_D3_out, TZD3_D3_out => TZD3_D3_out, work_D3_out => work_D3_out, ready_D3_out => ready_D3_out, TM_D3_out => TM_D3_out, RMS_D3_out => RMS_D3_out, DM_D3_out => DM_D3_out, KU_D4_out => KU_D4_out, TZN_D4_out => TZN_D4_out, UM_D4_out => UM_D4_out, KPM_D4_out => KPM_D4_out, TZV_D4_out => TZV_D4_out, KUD3_D4_out => KUD3_D4_out, TZD3_D4_out => TZD3_D4_out, work_D4_out => work_D4_out, ready_D4_out => ready_D4_out, avto_D4_out => avto_D4_out, TM_D4_out => TM_D4_out, RMS_D4_out => RMS_D4_out, DM_D4_out => DM_D4_out, KU_LK10_out => KU_LK10_out, TZ_LK10_out => TZ_LK10_out, tros_LK10_out => tros_LK10_out, shod_LK10_out => shod_LK10_out, ogr_LK10_out => ogr_LK10_out, avto_LK10_out => avto_LK10_out, ready_LK10_out => ready_LK10_out, work_LK10_out => work_LK10_out, KU_LK11_out => KU_LK11_out, TZ_LK11_out => TZ_LK11_out, tros_LK11_out => tros_LK11_out, shod_LK11_out => shod_LK11_out, ogr_LK11_out => ogr_LK11_out, avto_LK11_out => ato_LK11_out, ready_LK11_out => ready_LK11_out, work_LK11_out => work_LK11_out, KU_LK12_out => KU_LK12_out, TZ_LK12_out => TZ_LK12_out, tros_LK12_out => tros_LK12_out, shod_LK12_out => shod_LK12_out, ogr_LK12_out => ogr_LK12_out, avto_LK12_out => avto_LK12_out, ready_LK12_out => ready_LK12_out, work_LK12_out => work_LK12_out, KU_LK13_out => KU_LK13_out, TZ_LK13_out => TZ_LK13_out, tros_LK13_out => tros_LK13_out, shod_LK13_out => shod_LK13_out, ogr_LK13_out => ogr_LK13_out, avto_LK13_out => avto_LK13_out, ready_LK13_out => ready_LK13_out, work_LK13_out => work_LK13_out, avto_GR3_out => avto_GR3_out, KU_GR3_out => KU_GR3_out, TZ_GR3_out => TZ_GR3_out, ready_GR3_out => ready_GR3_out, work_GR3_out => work_GR3_out, STOP_GR3_out => STOP_GR3_out, KU_LK7_out => KU_LK7_out, TZ_LK7_out => TZ_LK7_out, tros_LK7_out => tros_LK7_out, shod_LK7_out => shod_LK7_out, ogr_LK7_out => ogr_LK7_out, avto_LK7_out => avto_LK7_out, ready_LK7_out => ready_LK7_out, work_LK7_out => work_LK7_out, KU_LK8_out => KU_LK8_out, TZ_LK8_out => TZ_LK8_out, tros_LK8_out => tros_LK8_out, shod_LK8_out => shod_LK8_out, ogr_LK8_out => ogr_LK8_out, avto_LK8_out => avto_LK8_out, ready_LK8_out => ready_LK8_out, work_LK8_out => work_LK8_out, KU_LK6_out => KU_LK6_out, TZ_LK6_out => TZ_LK6_out, tros_LK6_out => tros_LK6_out, shod_LK6_out => shod_LK6_out, ogr_LK6_out => ogr_LK6_out, avto_LK6_out => avto_LK6_out, ready_LK6_out => ready_LK6_out, work_LK6_out => work_LK6_out, KU_LK9_out => KU_LK9_out, TZ_LK9_out => TZ_LK9_out, tros_LK9_out => tros_LK9_out, shod_LK9_out => shod_LK9_out, ogr_LK9_out => ogr_LK9_out, avto_LK9_out => avto_LK9_out, ready_LK9_out => ready_LK9_out, work_LK9_out => work_LK9_out, KU_LP1_3_out => KU_LP1_3_out, in_020_out => in_020_out, in_040_out => in_040_out, in_020_4070_out => in_020_4070_out, TZ1_LP1_3_out => TZ1_LP1_3_out, TZ2_LP1_3_out => TZ2_LP1_3_out, TZ3_LP1_3_out => TZ3_LP1_3_out, PRO_LP1_3_out => PRO_LP1_3_out, avto_LP1_3_out => avto_LP1_3_out, ready_LP1_3_out => ready_LP1_3_out, work_LP1_3_out => work_LP1_3_out, stop2_LP1_3_out => stop2_LP1_3_out, avto_GR2_out => avto_GR2_out, KU_GR2_out => KU_GR2_out, TZ_GR2_out => TZ_GR2_out, ready_GR2_out => ready_GR2_out, work_GR2_out => work_GR2_out, STOP_GR2_out => STOP_GR2_out, KU_LK5_out => KU_LK5_out, TZ_LK5_out => TZ_LK5_out, tros_LK5_out => tros_LK5_out, shod_LK5_out => shod_LK5_out, ogr_LK5_out => ogr_LK5_out, avto_LK5_out => avto_LK5_out, ready_LK5_out => ready_LK5_out, work_LK5_out => work_LK5_out, KU_LK4_out => KU_LK4_out, TZ_LK4_out => TZ_LK4_out, tros_LK4_out => tros_LK4_out, shod_LK4_out => shod_LK4_out, avto_LK4_out => avto_LK4_out, ready_LK4_out => ready_LK4_out, work_LK4_out => work_LK4_out, MD3_LK4_out => MD3_LK4_out, avto_GR1_out => avto_GR1_out, KU_GR1_out => KU_GR1_out, TZ_GR1_out => TZ_GR1_out, ready_GR1_out => ready_GR1_out, work_GR1_out => work_GR1_out, STOP_GR1_out => STOP_GR1_out, KU_LK2_out => KU_LK2_out, TZ_LK2_out => TZ_LK2_out, tros_LK2_out => tros_LK2_out, shod_LK2_out => shod_LK2_out, ogr_LK2_out => ogr_LK2_out, avto_LK2_out => avto_LK2_out, ready_LK2_out => ready_LK2_out, work_LK2_out => work_LK2_out, KU_LK3_out => KU_LK3_out, TZ_LK3_out => TZ_LK3_out, tros_LK3_out => tros_LK3_out, shod_LK3_out => shod_LK3_out, ogr_LK3_out => ogr_LK3_out, avto_LK3_out => avto_LK3_out, ready_LK3_out => ready_LK3_out, work_LK3_out => work_LK3_out, avto_LP4_out => avto_LP4_out, ready_LP4_out => ready_LP4_out, work_LP4_out => work_LP4_out, MD2_LP4_out => MD2_LP4_out, output_Hz_LP4_out => output_Hz_LP4_out, avto_LP5_out => avto_LP5_out, ready_LP5_out => ready_LP5_out, work_LP5_out => work_LP5_out, STOP_LP5_out => STOP_LP5_out, MD2_LP5_out => MD2_LP5_out, output_Hz_LP5_out => output_Hz_LP5_out, avto_VP1_out => avto_VP1_out, ready_VP1_out => ready_VP1_out, work_VP1_out => work_VP1_out, STOP_VP1_out => STOP_VP1_out, KU_VP1_out => KU_VP1_out, TZ_VP1_out => TZ_VP1_out, avto_all_out => avto_all_out, pusk_out => pusk_out, PP1_out => PP1_out, LV_GR1_out => LV_GR1_out, LV_LK7_out => LV_LK7_out, LV_LK8_out => LV_LK8_out, LV_D2_out => LV_D2_out, lev_up_cyc_out => lev_up_cyc_out, pre_cyc_out => pre_cyc_out, ku_cyc_out => ku_cyc_out, tz_cyc_out => tz_cyc_out, ready_cyc_out => ready_cyc_out, work_cyc_out => work_cyc_out, shnek_up_cyc_out => shnek_up_cyc_out, avar_cyc_out => avar_cyc_out, gribok_out => gribok_out, TM_D3_word_out => TM_D3_word_out, TM_D4_word_out => TM_D4_word_out, avar_FC_lp5_out => avar_FC_LP5_out, lev_down_cyc_out => lev_down_cyc_out) => KU_D2_out
NETWORK 62
	*
		EN --- signals1:bool_to(pusk_LAN_LP4: pusk_LAN_LP4, stop_LAN_LP4: stop_LAN_LP4, pusk_LAN_LP5: pusk_LAN_LP5, stop_LAN_LP5: stop_LAN_LP5, pusk_LAN_VP1: pusk_LAN_VP1, stop_LAN_VP1: stop_LAN_VP1, pusk_lan_LK10: pusk_lan_LK10, pusk_lan_LK11: pusk_lan_LK11, pusk_lan_LK12: pusk_lan_LK12, pusk_lan_LK13: pusk_lan_LK13, pusk_lan_GR3: pusk_lan_GR3, pusk_lan_LK7: pusk_lan_LK7, pusk_lan_LK8: pusk_lan_LK8, pusk_lan_LK6: pusk_lan_LK6, pusk_lan_LK9: pusk_lan_LK9, pusk_lan_LP1_3: pusk_lan_LP1_3, pusk_lan_GR2: pusk_lan_GR2, pusk_lan_LK5: pusk_lan_LK5, pusk_lan_LK4: pusk_lan_LK4, pusk_lan_LK3: pusk_lan_LK3, pusk_lan_GR1: pusk_lan_GR1, pusk_lan_LK2: pusk_lan_LK2, stop_lan_LK10: stop_lan_LK10, stop_lan_LK11: stop_lan_LK11, stop_lan_LK12: stop_lan_LK12, stop_lan_LK13: stop_lan_LK13, stop_lan_GR3: stop_lan_GR3, stop_lan_LK7: stop_lan_LK7, stop_lan_LK8: stop_lan_LK8, stop_lan_LK6: stop_lan_LK6, stop_lan_LK9: stop_lan_LK9, stop_lan_LP1_3: stop_lan_LP1_3, stop_lan_GR2: stop_lan_GR2, stop_lan_LK5: stop_lan_LK5, stop_lan_LK4: stop_lan_LK4, stop_lan_LK3: stop_lan_LK3, stop_lan_GR1: stop_lan_GR1, stop_lan_LK2: stop_lan_LK2, stop_LAN_D3: stop_LAN_D3, stop_LAN_D4: stop_LAN_D4, pusk_lan_D2: pusk_LAN_D2, stop_lan_D2: stop_LAN_D2, pusk_lan_D3: pusk_LAN_D3, pusk_lan_D4: pusk_LAN_D4, pusk_lan_cyclone: pusk_lan_cyclone, stop_lan_cyclone: stop_lan_cyclone, tros_self_lk10_in: tros_self_lk10, shod_self_lk10_in: shod_self_lk10, ogr_self_lk10_in: ogr_self_lk10, vl_self_lk10_in: vl_self_lk10, tros_self_lk11_in: tros_self_lk11, shod_self_lk11_in: shod_self_lk11, ogr_self_lk11_in: ogr_self_lk11, vl_self_lk11_in: vl_self_lk11, tros_self_lk12_in: tros_self_lk12, shod_self_lk12_in: shod_self_lk12, ogr_self_lk12_in: ogr_self_lk12, vl_self_lk12_in: vl_self_lk12, tros_self_lk13_in: tros_self_lk13, shod_self_lk13_in: shod_self_lk13, ogr_self_lk13_in: ogr_self_lk13, vl_self_lk13_in: vl_self_lk13, tros_self_lk7_in: tros_self_lk7, shod_self_lk7_in: shod_self_lk7, ogr_self_lk7_in: ogr_self_lk7, vl_self_lk7_in: vl_self_lk7, tros_self_lk8_in: tros_self_lk8, shod_self_lk8_in: shod_self_lk8, ogr_self_lk8_in: ogr_self_lk8, vl_self_lk8_in: vl_self_lk8, tros_self_lk6_in: tros_self_lk6, shod_self_lk6_in: shod_self_lk6, ogr_self_lk6_in: ogr_self_lk6, vl_self_lk6_in: vl_self_lk6, tros_self_lk9_in: tros_self_lk9, shod_self_lk9_in: shod_self_lk9, ogr_self_lk9_in: ogr_self_lk9, vl_self_lk9_in: vl_self_lk9, vl_self_lp1_3_in: vl_self_lp1_3, tros_self_lk5_in: tros_self_lk5, shod_self_lk5_in: shod_self_lk5, ogr_self_lk5_in: ogr_self_lk5, vl_self_lk5_in: vl_self_lk5, tros_self_lk4_in: tros_self_lk4, shod_self_lk4_in: shod_self_lk4, vl_self_lk4_in: vl_self_lk4, tros_self_lk3_in: tros_self_lk3, shod_self_lk3_in: shod_self_lk3, ogr_self_lk3_in: ogr_self_lk3, vl_self_lk3_in: vl_self_lk3, tros_self_lk2_in: tros_self_lk2, shod_self_lk2_in: shod_self_lk2, ogr_self_lk2_in: ogr_self_lk2, vl_self_lk2_in: vl_self_lk2, revers_in: revers, vl_self_lp4_in: vl_self_lp4, vl_self_lp5_in: vl_self_lp5, pusk_shnek_razg_in: pusk_shnek_razg, stop_shnek_razg_in: stop_shnek_razg, pusk_cyc_cleen_in: pusk_cleen_lan, stop_cyc_cleen_in: stop_cleen_lan, stop_LAN_LP4_out => stop_LAN_LP4_out, pusk_LAN_LP5_out => pusk_LAN_LP5_out, stop_LAN_LP5_out => stop_LAN_LP5_out, pusk_LAN_VP1_out => pusk_LAN_VP1_out, stop_LAN_VP1_out => stop_LAN_VP1_out, pusk_lan_LK10_out => pusk_lan_LK10_out, pusk_lan_LK11_out => pusk_lan_LK11_out, pusk_lan_LK12_out => pusk_lan_LK12_out, pusk_lan_LK13_out => pusk_lan_LK13_out, pusk_lan_GR3_out => pusk_lan_GR3_out, pusk_lan_LK7out => pusk_lan_LK7_out, pusk_lan_LK8_out => pusk_lan_LK8_out, pusk_lan_LK6_out => pusk_lan_LK6_out, pusk_lan_LK9_out => pusk_lan_LK9_out, pusk_lan_LP1_3_out => pusk_lan_LP1_3_out, pusk_lan_GR2_out => pusk_lan_GR2_out, pusk_lan_LK5_out => pusk_lan_LK5_out, pusk_lan_LK4_out => pusk_lan_LK4_out, pusk_lan_LK3_out => pusk_lan_LK3_out, pusk_lan_GR1_out => pusk_lan_GR1_out, pusk_lan_LK2_out => pusk_lan_LK2_out, stop_lan_LK10_out => stop_lan_LK10_out, stop_lan_LK11_out => stop_lan_LK11_out, stop_lan_LK12_out => stop_lan_LK12_out, stop_lan_LK13_out => stop_lan_LK13_out, stop_lan_GR3_out => stop_lan_GR3_out, stop_lan_LK7_out => stop_lan_LK7_out, stop_lan_LK8_out => stop_lan_LK8_out, stop_lan_LK6_out => stop_lan_LK6_out, stop_lan_LK9_out => stop_lan_LK9_out, stop_lan_LP1_3_out => stop_lan_LP1_3_out, stop_lan_GR2_out => stop_lan_GR2_out, stop_lan_LK5_out => stop_lan_LK5_out, stop_lan_LK4_out => stop_lan_LK4_out, stop_lan_LK3_out => stop_lan_LK3_out, stop_lan_GR1_out => stop_lan_GR1_out, stop_lan_LK2_out => stop_lan_LK2_out, stop_LAN_D3_out => stop_LAN_D3_out, stop_LAN_D4_out => stop_LAN_D4_out, pusk_lan_D2_out => pusk_LAN_D2_out, stop_lan_D2_out => stop_LAN_D2_out, pusk_lan_D3_out => pusk_LAN_D3_out, pusk_lan_D4_out => pusk_LAN_D4_out, pusk_lan_cyclone_out => pusk_lan_cyclone_out, stop_lan_cyclone_out => stop_lan_cyclone_out, tros_self_lk10_out => tros_self_lk10_out, shod_self_lk10_out => shod_self_lk10_out, ogr_self_lk10_out => ogr_self_lk10_out, vl_self_lk10_out => vl_self_lk10_out, tros_self_lk11_out => tros_self_lk11_out, shod_self_lk11_out => shod_self_lk11_out, ogr_self_lk11_out => ogr_self_lk11_out, vl_self_lk11_out => vl_self_lk11_out, tros_self_lk12_out => tros_self_lk12_out, shod_self_lk12_out => shod_self_lk12_out, ogr_self_lk12_out => ogr_self_lk12_out, vl_self_lk12_out => vl_self_lk12_out, tros_self_lk13_out => tros_self_lk13_out, shod_self_lk13_out => shod_self_lk13_out, ogr_self_lk13_out => ogr_self_lk13_out, vl_self_lk13_out => vl_self_lk13_out, tros_self_lk7_out => tros_self_lk7_out, shod_self_lk7_out => shod_self_lk7_out, ogr_self_lk7_out => ogr_self_lk7_out, vl_self_lk7_out => vl_self_lk7_out, tros_self_lk8_out => tros_self_lk8_out, shod_self_lk8_out => shod_self_lk8_out, ogr_self_lk8_out => ogr_self_lk8_out, vl_self_lk8_out => vl_self_lk8_out, tros_self_lk6_out => tros_self_lk6_out, shod_self_lk6_out => shod_self_lk6_out, ogr_self_lk6_out => ogr_self_lk6_out, vl_self_lk6_out => vl_self_lk6_out, tros_self_lk9_out => tros_self_lk9_out, shod_self_lk9_out => shod_self_lk9_out, ogr_self_lk9_out => ogr_self_lk9_out, vl_self_lk9_out => vl_self_lk9_out, vl_self_lp1_3_out => vl_self_lp1_3_out, tros_self_lk5_out => tros_self_lk5_out, shod_self_lk5_out => shod_self_lk5_out, ogr_self_lk5_out => ogr_self_lk5_out, vl_self_lk5_out => vl_self_lk5_out, tros_self_lk4_out => tros_self_lk4_out, shod_self_lk4_out => shod_self_lk4_out, vl_self_lk4_out => vl_self_lk4_out, tros_self_lk3_out => tros_self_lk3_out, shod_self_lk3_out => shod_self_lk3_out, ogr_self_lk3_out => ogr_self_lk3_out, vl_self_lk3_out => vl_self_lk3_out, tros_self_lk2_out => tros_self_lk2_out, shod_self_lk2_out => shod_self_lk2_out, ogr_self_lk2_out => ogr_self_lk2_out, vl_self_lk2_out => vl_self_lk2_out, revers_out => revers_out, vl_self_lp4_out => vl_self_lp4_out, vl_self_lp5_out => vl_self_lp5_out, pusk_shnek_razg_out => pusk_shnek_razg_out, stop_shnek_razg_out => stop_shnek_razg_out, pusk_cyc_cleen_out => cyc_cleen_pusk, stop_cyc_cleen_out => cyc_cleen_stop) => pusk_LAN_LP4_out
NETWORK 63
	*
		EN --- alarm:alarm(adress_in_rs2: adr_dev_rs2, error_81_in_rs2: err_dev_rs2, adress_in_rs1: adr_dev_rs1, error_81_in_rs1: err_dev_rs1, err_LK11 => e_LK11_out, err_LK12 => e_LK12_out, err_LK13 => e_LK13_out, err_GR3 => e_GR3_out, err_LK7 => e_LK7_out, err_LK8 => e_LK8_out, err_LK6 => e_LK6_out, err_LK9 => e_LK9_out, err_LP1_3_mod1 => e_LP13mod1_out, err_LP1_3_mod2 => e_LP13mod2_out, err_GR2 => e_GR2_out, err_LK5 => e_LK5_out, err_LP4 => e_LP4_out, err_LP5 => e_LP5_out, err_LK4 => e_LK4_out, err_GR1 => e_GR1_out, err_LK2 => e_LK2_out, err_LK3 => e_LK3_out, err_VP1 => e_VP1_out, err_D3_mod1 => e_D3mod1_out, err_D3_mod2 => e_D3mod2_out, err_D4_mod1 => e_D4mod1_out, err_D4_mod2 => e_D4mod2_out, err_D2 => e_D2_out, err_cyc1 => e_cyc1_out, err_cyc2 => e_cyc2_out, err_lp4_temp => e_lp4_temp_out, err_d3_temp => e_d3_temp_out, err_d4_temp => e_d4_temp_out, err_vp1_temp => e_vp1_temp_out) => e_LK10_out
		EN --- alarm_all:alarm_all(err_LK10: e_LK10_out, err_LK11: e_LK11_out, err_LK12: e_LK12_out, err_LK13: e_LK13_out, err_GR3: e_GR3_out, err_LK7: e_LK7_out, err_LK8: e_LK8_out, err_LK6: e_LK6_out, err_LK9: e_LK9_out, err_LP1_3_mod1: e_LP13mod1_out, err_LP1_3_mod2: e_LP13mod2_out, err_GR2: e_GR2_out, err_LK5: e_LK5_out, err_LP4: e_LP4_out, err_LP5: e_LP5_out, err_LK4: e_LK4_out, err_GR1: e_GR1_out, err_LK2: e_LK2_out, err_LK3: e_LK3_out, err_VP1: e_VP1_out, err_D3_mod1: e_D3mod1_out, err_D3_mod2: e_D3mod2_out, err_D4_mod1: e_D4mod1_out, err_D4_mod2: e_D4mod2_out, err_D2: e_D2_out, err_cyc1: e_cyc1_out, err_cyc2: e_cyc2_out, err_lp4_temp: e_lp4_temp_out, err_d3_temp: e_d3_temp_out, err_d4_temp: e_d4_temp_out, err_vp1_temp: e_vp1_temp_out) => moduls_out
_END_LD_
(* the same logic as Structured Text *)
(* Network 1: Фиксация пуска для SCADA-системы *)
pusk_lan := (pusk_sys AND avto_all OR pusk_lan) AND NOT stop_DDD AND NOT gribok;
(* Network 2: Пуск только по готовностям всех шкафов *)
pusk := pusk_sys AND avto_all AND ready_D2 AND ready_D3 AND (ready_D4 OR in_040) AND ready_LK10 AND ready_LK11 AND (ready_LK12 OR NOT current_value_lk_glob) AND ready_LK13 AND ready_GR3 AND (ready_LK7 OR in_040) AND ready_LK8 AND ready_LK9 AND (ready_LK6 OR in_020) AND ready_LP1_3 AND ready_GR2 AND ready_LK5 AND ready_LP4 AND (ready_LP5 OR in_040) AND ready_GR1 AND ready_LK2 AND ready_VP1 AND ready_LK3;
(* Network 3: Остановка всех агрегатов по втором нажатии кнопки "стоп" *)
stop(CU := stop_sys, RESET := stop_DDD OR pusk_sys OR ruchnoe_all, PV := 2);
stop_all := stop.Q;
(* Network 4: Остановка дробилок по третьему нажатию кнопки "стоп" *)
stop_Drob(CU := stop_sys, RESET := stop_DDD OR pusk_sys, PV := 3);
stop_D2 := stop_Drob.Q;
(* Network 5 *)
cyclone(stop := stop_DDD, grib := gribok, pusk_LAN := pusk_lan_cyclone_out, stop_lan := stop_lan_cyclone_out, level := lev_up_cyc, KU := ku_cyc, TZ := tz_cyc, skvaj := skvaj_in, switch := revers_out, err := e_cyc1_out OR e_cyc2_out, pusk_shnek_lan := pusk_shnek_razg_out, stop_shnek_lan := stop_shnek_razg_out, in_time := in_time_shake, time_run := time_run, time_stop := time_stop, cleen_in_pusk := cyc_cleen_pusk, cleen_in_stop := cyc_cleen_stop);
ve1_out := cyclone.VE_1;
ve2_out := cyclone.VE_2;
ve3_out := cyclone.VE_3;
ve4_out := cyclone.VE_4;
ve5_out := cyclone.VE_5;
ve6_out := cyclone.VE_6;
ve7_out := cyclone.VE_7;
ve8_out := cyclone.VE_8;
shnek_up_cyc := cyclone.shnek_up;
ready_cyc := cyclone.ready;
work_cyc := cyclone.work;
avar_cyc := cyclone.avar;
shnek_razg := cyclone.shnek_razg;
prom_cleen_out := cyclone.prom_cleen_word;
vent_pump_cyc := cyclone.vent;
(* Network 6 *)
km_byte_cyc := PACK(shnek_razg, vent_pump_cyc, shnek_up_cyc, FALSE, FALSE, FALSE, FALSE, FALSE);
(* Network 7: Блок управления дробилкой Д2 *)
D2(pusk := pusk, KUD2 := KU_D2, RMS2_2 := RMS2_2, RD2 := RD2_D2, TZD2 := TZD2, avto := avto_D2, GRIB := gribok, stop_s := stop_D2, ruchnoe := ruchnoe_all, pusk_LAN := pusk_LAN_D2_out, stop_LAN := stop_LAN_D2_out, err := e_D2_out);
work_D2 := D2.work;
KM2_D2 := D2.KM2;
KM3_D2 := D2.KM3;
stop_D3 := D2.stop_D3D4;
avar_D2 := D2.avar;
ready_D2 := D2.ready;
(* Network 8: Блок управления битовой маской выходов модуля расширения в шкафу управления Д2 *)
KM_D2_byte := PACK(FALSE, KM2_D2, FALSE, KM3_D2, FALSE, FALSE, FALSE, FALSE);
(* Network 9: Блок управления дробилкой Д3 *)
D3(pusk := pusk, KU := KU_D3, TZN := TZN_D3, KPM := KPM_D3, TZV := TZV_D3, KUD3 := KUD3_D3, TZD3 := TZD3_D3, RD3 := RD3_D3, TM := TM_D3, RMS := RMS_D3, avto_in := avto_D3, GRIB := gribok, work_D2_D3 := work_D2, stop_in := stop_D2, ruchnoe := ruchnoe_all, pusk_LAN := pusk_LAN_D3_out, stop_LAN := stop_LAN_D3_out, err := e_D3mod1_out OR e_D3mod2_out, UM := UM_D3);
KM2_D3 := D3.KM2;
KM3_D3 := D3.KM3;
ready_D3 := D3.ready;
nasos_D3 := D3.nasos;
vent_D3 := D3.vent;
ten_D3 := D3.ten;
work_D3 := D3.work;
out_avto_D3 := D3.avto;
avar_D3 := D3.avar;
stop_D4 := D3.stop_D3D4;
TM_D3_bool := D3.tm_ins;
KM1_D3 := D3.KM1;
(* Network 10: Блок управления битовой маской выходов модуля расширения в шкафу управления Д4 *)
D3_mod1_byte := PACK(out_avto_D3, nasos_D3, vent_D3, ten_D3, FALSE, FALSE, FALSE, FALSE);
D3_mod2_byte := PACK(FALSE, KM1_D3, KM2_D3, KM3_D3, FALSE, FALSE, FALSE, FALSE);
(* Network 11: Блок управления дробилкой Д4 *)
D4(pusk := pusk, KU := KU_D4, TZN := TZN_D4, KPM := KPM_D4, TZV := TZV_D4, KUD3 := KUD3_D4, TZD3 := TZD3_D4, RD3 := RD3_D4, TM := TM_D4, RMS := RMS_D4, avto_in := avto_D4, GRIB := gribok, work_D2_D3 := work_D3, stop_in := stop_D4, ruchnoe := ruchnoe_all, ins_0_40 := in_040, pusk_LAN := pusk_LAN_D4_out, stop_LAN := stop_LAN_D4_out, err := e_D4mod1_out OR e_D4mod2_out, UM := UM_D4);
KM2_D4 := D4.KM2;
KM3_D4 := D4.KM3;
ready_D4 := D4.ready;
nasos_D4 := D4.nasos;
vent_D4 := D4.vent;
ten_D4 := D4.ten;
work_D4 := D4.work;
out_avto_D4 := D4.avto;
avar_D4 := D4.avar;
stop_DDD := D4.stop_D3D4;
TM_D4_bool := D4.tm_ins;
KM1_D4 := D4.KM1;
(* Network 12: Блок управления битовой маской выходов модуля расширения в шкафу управления Д4 *)
D4_mod1_byte := PACK(out_avto_D4, nasos_D4, vent_D4, ten_D4, FALSE, FALSE, FALSE, FALSE);
D4_mod2_byte := PACK(FALSE, KM1_D4, KM2_D4, KM3_D4, FALSE, FALSE, FALSE, FALSE);
(* Network 13: Подтверждение работы дробилок Д2-Д4 и разрешение на пуск следующей ступени агрегатов *)
work_level_10 := work_D2 AND work_D3 AND (work_D4 OR in_040);
(* Network 14: Проверка готовностей ленточных конвееров ЛК10-ЛК13. После пуска всех агрегатов этой ступени, / промежуточное реле самоподхвата разрывается для защиты от повторного пуска *)
prom1 := (pusk AND ready_LK10 AND ready_LK11 AND ready_LK13 OR prom1 AND NOT work_level_1 AND NOT avar_LK10 AND NOT avar_LK11 AND NOT avar_LK13) AND NOT STOP_SYS AND NOT stop_lan_LK10_out AND NOT stop_lan_LK11_out AND NOT stop_lan_LK13_out;
(* Network 15: Блок управления ленточным конвеером ЛК-10 *)
ton_LK10(IN := work_level_10, PT := t#1s);
LK10(pusk := ton_LK10.Q AND avto_all AND prom1, avto := avto_LK10, KU := KU_LK10, TZ := TZ_LK10, tros := tros_LK10, shod := shod_LK10, ogr := ogr_LK10, VL := bool_Vl_LK10, P := P_LK10, GRIB := gribok, stop_s := stop_all, ruchnoe := ruchnoe_all, pusk_LAN := pusk_lan_LK10_out, stop_LAN := stop_lan_LK10_out, err := e_LK10_out, tros_self := tros_self_lk10_out, shod_self := shod_self_lk10_out, ogr_self := ogr_self_lk10_out, pusk_sys_ins := PUSK_SYS);
ready_LK10 := LK10.ready;
work_LK10 := LK10.work;
avar_LK10 := LK10.avar;
avar_vl_lk10 := LK10.avar_vl;
KM1_LK10 := LK10.KM;
(* Network 16: Блок управления ленточным конвеером ЛК-11 *)
ton_lk11(IN := work_LK10, PT := t#1s);
LK11(pusk := ton_lk11.Q AND avto_all AND prom1, avto := avto_LK11, KU := KU_LK11, TZ := TZ_LK11, tros := tros_LK11, shod := shod_LK11, ogr := ogr_LK11, VL := bool_Vl_LK11, P := P_LK11, GRIB := gribok, stop_s := stop_all, ruchnoe := ruchnoe_all, pusk_LAN := pusk_lan_LK11_out, stop_LAN := stop_lan_LK11_out, err := e_LK11_out, tros_self := tros_self_lk11_out, shod_self := shod_self_lk11_out, ogr_self := ogr_self_lk11_out, pusk_sys_ins := PUSK_SYS);
ready_LK11 := LK11.ready;
work_LK11 := LK11.work;
avar_LK11 := LK11.avar;
avar_vl_lk11 := LK11.avar_vl;
KM1_LK11 := LK11.KM;
(* Network 17: Блок управления ленточным конвеером ЛК-12 *)
ton_lk12(IN := work_LK11, PT := t#1s);
LK12(pusk := ton_lk12.Q AND avto_all AND prom1, avto := avto_LK12, KU := KU_LK12, TZ := TZ_LK12, tros := tros_LK12, shod := shod_LK12, ogr := ogr_LK12, VL := bool_Vl_LK12, P := P_LK12, GRIB := gribok, stop_s := stop_all, ruchnoe := ruchnoe_all, pusk_LAN := pusk_lan_LK12_out, stop_LAN := stop_lan_LK12_out, err := e_LK12_out, tros_self := tros_self_lk12_out, shod_self := shod_self_lk12_out, ogr_self := ogr_self_lk12_out, pusk_sys_ins := PUSK_SYS, switcher_in := lk12_switcher, current_value_lk12_in := current_value_lk_glob);
ready_LK12 := LK12.ready;
work_LK12 := LK12.work;
avar_LK12 := LK12.avar;
avar_vl_lk12 := LK12.avar_vl;
current_value_lk_glob := LK12.current_value_lk12_out;
KM1_LK12 := LK12.KM;
(* Network 18: Блок управления ленточным конвеером ЛК-13 *)
ton_lk13(IN := work_LK11, PT := t#1s);
LK13(pusk := ton_lk13.Q AND avto_all AND prom1, avto := avto_LK13, KU := KU_LK13, TZ := TZ_LK13, tros := tros_LK13, shod := shod_LK13, ogr := ogr_LK13, VL := bool_Vl_LK13, P := P_LK13, GRIB := gribok, stop_s := stop_all, ruchnoe := ruchnoe_all, pusk_LAN := pusk_lan_LK13_out, stop_LAN := stop_lan_LK13_out, err := e_LK13_out, tros_self := tros_self_lk13_out, shod_self := shod_self_lk13_out, ogr_self := ogr_self_lk13_out, pusk_sys_ins := PUSK_SYS);
ready_LK13 := LK13.ready;
work_LK13 := LK13.work;
avar_LK13 := LK13.avar;
avar_vl_lk13 := LK13.avar_vl;
KM1_LK13 := LK13.KM;
(* Network 19: Подтверждение работы конвееров ЛК10-ЛК13 и разрешение на пуск следующей ступени агрегатов *)
work_level_1 := work_LK10 AND work_LK11 AND work_LK13;
(* Network 20: Определить, какой из конвееров первой ветки остановился *)
stop_vl_lv1 := avar_vl_lk10 OR avar_vl_lk11 OR avar_vl_lk13;
(* Network 21: Проверка готовности грохота ГР3. После пуска агрегата, / промежуточное реле самоподхвата разрывается для защиты от повторного пуска *)
prom2 := (pusk AND ready_GR3 OR prom2 AND NOT work_GR3 AND NOT avar_GR3) AND NOT STOP_SYS AND NOT stop_lan_GR3_out;
(* Network 22: Блок управления грохотом ГР3 *)
ton_GR3(IN := work_level_1, PT := t#1s);
GR3(pusk := ton_GR3.Q AND avto_all AND prom2, avto := avto_GR3, KU := KU_gr3, TZ := TZ_gr3, P := p_gr3, STOP := STOP_GR3, GRIB := gribok, stop_s := stop_all, ruchnoe := ruchnoe_all, pusk_LAN := pusk_lan_GR3_out, stop_LAN := stop_lan_GR3_out, err := e_GR3_out);
ready_GR3 := GR3.ready;
work_GR3 := GR3.work;
avar_GR3 := GR3.avar;
KM1_GR3 := GR3.KM;
(* Network 23: Подтверждение работы ступени №1 и грохота, и разрешение на пуск следующей ступени агрегатов *)
work_level_2 := work_level_1 AND work_GR3;
(* Network 24: Проверка готовностей ленточных конвееров ЛК6,ЛК7-ЛК9. После пуска всех агрегатов этой ступени, / промежуточное реле самоподхвата разрывается для защиты от повторного пуска *)
prom3 := (pusk AND (ready_LK7 OR in_040) AND ready_LK8 AND ready_LK9 AND (ready_LK6 OR in_020) OR prom3 AND NOT work_level_3 AND NOT avar_LK7 AND NOT avar_LK8 AND NOT avar_LK6 AND NOT avar_LK9) AND NOT STOP_SYS AND NOT stop_lan_LK7_out AND NOT stop_lan_LK8_out AND NOT stop_lan_LK6_out AND NOT stop_lan_LK9_out;
(* Network 25: Блок управления ленточным конвеером ЛК-7 *)
ton_LK7(IN := work_GR3, PT := t#10s);
LK7(pusk := ton_LK7.Q AND avto_all AND prom3, avto := avto_LK7, KU := KU_LK7, TZ := TZ_LK7, tros := tros_LK7, shod := shod_LK7, ogr := ogr_LK7, VL := bool_Vl_LK7, P := P_LK7, in_020 := in_040, stop_s := stop_all, GRIB := gribok, ruchnoe := ruchnoe_all, pusk_LAN := pusk_lan_LK7_out, stop_LAN := stop_lan_LK7_out, err := e_LK7_out, tros_self := tros_self_lk7_out, shod_self := shod_self_lk7_out, ogr_self := ogr_self_lk7_out, pusk_sys_ins := PUSK_SYS);
ready_LK7 := LK7.ready;
work_LK7 := LK7.work;
avar_LK7 := LK7.avar;
avar_vl_lk7 := LK7.avar_vl;
KM1_LK7 := LK7.KM;
(* Network 26: Блок управления ленточным конвеером ЛК-8 *)
ton_LK8(IN := work_LK7, PT := t#1s);
ton_LK81(IN := work_GR3 AND in_040, PT := t#10s);
LK8(pusk := (ton_LK8.Q OR ton_LK81.Q) AND avto_all AND prom3, avto := avto_LK8, KU := KU_LK8, TZ := TZ_LK8, tros := tros_LK8, shod := shod_LK8, ogr := ogr_LK8, VL := bool_Vl_LK8, P := P_LK8, GRIB := stop_all, stop_s := gribok, ruchnoe := ruchnoe_all, pusk_LAN := pusk_lan_LK8_out, stop_LAN := stop_lan_LK8_out, err := e_LK8_out, tros_self := tros_self_lk8_out, shod_self := shod_self_lk8_out, ogr_self := ogr_self_lk8_out, pusk_sys_ins := PUSK_SYS);
ready_LK8 := LK8.ready;
work_LK8 := LK8.work;
avar_LK8 := LK8.avar;
avar_vl_lk8 := LK8.avar_vl;
KM1_LK8 := LK8.KM;
(* Network 27: Блок управления ленточным конвеером ЛК-6 *)
ton_LK6(IN := work_LK8, PT := t#1s);
LK6(pusk := ton_LK6.Q AND avto_all AND prom3, avto := avto_LK6, KU := KU_LK6, TZ := TZ_LK6, tros := tros_LK6, shod := shod_LK6, ogr := ogr_LK6, VL := bool_Vl_LK6, P := P_LK6, in_020 := in_020, stop_s := stop_all, GRIB := gribok, ruchnoe := ruchnoe_all, pusk_LAN := pusk_lan_LK6_out, stop_LAN := stop_lan_LK6_out, err := e_LK6_out, tros_self := tros_self_lk6_out, shod_self := shod_self_lk6_out, ogr_self := ogr_self_lk6_out, pusk_sys_ins := PUSK_SYS);
ready_LK6 := LK6.ready;
work_LK6 := LK6.work;
avar_LK6 := LK6.avar;
avar_vl_lk6 := LK6.avar_vl;
KM1_LK6 := LK6.KM;
(* Network 28: Блок управления ленточным конвеером ЛК-9 *)
ton_LK9(IN := work_LK6 OR in_020 AND work_LK8, PT := t#1s);
LK9(pusk := ton_LK9.Q AND avto_all AND prom3, avto := avto_LK9, KU := KU_LK9, TZ := TZ_LK9, tros := tros_LK9, shod := shod_LK9, ogr := ogr_LK9, VL := bool_Vl_LK9, P := P_LK9, GRIB := gribok, stop_s := stop_all, ruchnoe := ruchnoe_all, pusk_LAN := pusk_lan_LK9_out, stop_LAN := stop_lan_LK9_out, err := e_LK9_out, tros_self := tros_self_lk9_out, shod_self := shod_self_lk9_out, ogr_self := ogr_self_lk9_out, pusk_sys_ins := PUSK_SYS);
ready_LK9 := LK9.ready;
work_LK9 := LK9.work;
avar_LK9 := LK9.avar;
avar_vl_lk9 := LK9.avar_vl;
KM1_LK9 := LK9.KM;
(* Network 29 *)
stop_vl_lv2 := avar_vl_lk7 OR avar_vl_lk8 OR avar_vl_lk6 OR avar_vl_lk9 OR stop_vl_lv1;
(* Network 30: Подтверждение работы конвееров ЛК6,ЛК7-ЛК9 и разрешение на пуск следующей ступени агрегатов *)
work_level_3 := (work_LK7 OR in_040) AND work_LK8 AND (work_LK6 OR in_020) AND work_LK9;
(* Network 31: Проверка готовности ленточного питателя ЛП1-ЛП3. После пуска всех агрегатов этой ступени, / промежуточное реле самоподхвата разрывается для защиты от повторного пуска *)
prom4 := (pusk AND ready_LP1_3 OR prom4 AND NOT work_LP1_3 AND NOT avar_LP1_3) AND NOT STOP_SYS AND NOT stop_lan_LP1_3_out;
(* Network 32: Блок управления ленточным питетелем ЛП1-ЛП3 *)
ton_LP1_3(IN := work_LK9, PT := t#1s);
LP1_3(pusk_sys := ton_LP1_3.Q AND avto_all AND prom4, Vl1 := TRUE, Vl2 := TRUE, Vl3 := TRUE, in_020 := in_020, in_040 := in_040, in_020_4070 := in_020_4070, KU := KU_LP1_3, TZ1 := TZ1_LP1_3, TZ2 := TZ2_LP1_3, TZ3 := TZ3_LP1_3, PRO := PRO_LP1_3, avto := avto_LP1_3, P := P_LP1_3, stop2 := stop2_LP1_3, GRIB := gribok, stop_s := stop_all, ruchnoe := ruchnoe_all, pusk_LAN := pusk_lan_LP1_3_out, stop_LAN := stop_lan_LP1_3_out, err := e_LP13mod1_out OR e_LP13mod2_out, pusk_sys_ins := PUSK_SYS);
KM2_LP1_3 := LP1_3.KM2;
KM4_LP1_3 := LP1_3.KM4;
KM5_LP1_3 := LP1_3.KM5;
KM3_LP1_3 := LP1_3.KM3;
ready_LP1_3 := LP1_3.ready;
work_LP1_3 := LP1_3.work;
avar_LP1_3 := LP1_3.avar;
avar_vl_lp1_3 := LP1_3.avar_vl;
KM1_LP1_3 := LP1_3.KM1;
(* Network 33: Блок управления битовой маской выходов модуля расширения в шкафу управления ЛП1-ЛП3 *)
KM2345_LP1_3_byte := PACK(KM2_LP1_3, KM3_LP1_3, KM4_LP1_3, KM5_LP1_3, FALSE, FALSE, FALSE, FALSE);
(* Network 34: Проверка готовности грохота ГР2. После пуска всех агрегатов этой ступени, / промежуточное реле самоподхвата разрывается для защиты от повторного пуска *)
prom5 := (pusk AND ready_GR2 OR prom5 AND NOT avar_GR2 AND NOT work_GR2) AND NOT STOP_SYS AND NOT stop_lan_GR2_out;
(* Network 35: Блок управления грохотом ГР2 *)
ton_GR2(IN := work_LP1_3, PT := t#1s);
GR2(pusk := ton_GR2.Q AND avto_all AND prom5, avto := avto_GR2, KU := KU_GR2, TZ := TZ_GR2, P := P_GR2, STOP := STOP_GR2, stop_sys := gribok, GRIB := stop_all, stop_lv := work_LP1_3, ruchnoe := ruchnoe_all, pusk_LAN := pusk_lan_GR2_out, stop_LAN := stop_lan_GR2_out, err := e_GR2_out);
ready_GR2 := GR2.ready;
work_GR2 := GR2.work;
avar_GR2 := GR2.avar;
KM1_GR2 := GR2.KM;
(* Network 36: Подтверждение работы ГР2, ЛП1-ЛП3 и разрешение на пуск следующей ступени агрегатов *)
work_level_4 := work_level_3 AND work_GR2;
(* Network 37 *)
stop_vl_lv2 := avar_vl_lk7 OR avar_vl_lk8 OR avar_vl_lk6 OR avar_vl_lk9 OR avar_vl_lp1_3 OR stop_vl_lv1;
(* Network 38: Проверка готовности ленточного конвеера ЛК5. После пуска всех агрегатов этой ступени, / промежуточное реле самоподхвата разрывается для защиты от повторного пуска *)
prom6 := (pusk AND ready_LK5 OR prom6 AND NOT avar_LK5 AND NOT work_LK5) AND NOT STOP_SYS AND NOT stop_lan_LK5_out;
(* Network 39: Блок управления ленточного конвеера ЛК5 *)
ton_LK5(IN := work_GR2, PT := t#10s);
LK5(pusk := ton_LK5.Q AND avto_all AND prom6, avto := avto_LK5, KU := KU_LK5, TZ := TZ_LK5, tros := tros_LK5, shod := shod_LK5, ogr := ogr_LK5, VL := bool_Vl_LK5, P := P_LK5, GRIB := gribok, stop_s := stop_all, ruchnoe := ruchnoe_all, pusk_LAN := pusk_lan_LK5_out, stop_LAN := stop_lan_LK5_out, err := e_LK5_out, tros_self := tros_self_lk5_out, shod_self := shod_self_lk5_out, ogr_self := ogr_self_lk5_out, pusk_sys_ins := PUSK_SYS);
ready_LK5 := LK5.ready;
work_LK5 := LK5.work;
avar_LK5 := LK5.avar;
avar_vl_lk5 := LK5.avar_vl;
KM1_LK5 := LK5.KM;
(* Network 40: Подтверждение работы дробилки Д3 и ленточного конвеера ЛК5, и разрешение на пуск следующей ступени агрегатов *)
work_level_6 := work_D3 AND work_LK5 AND work_level_2 AND work_level_4;
(* Network 41: Подтверждение работы дробилки Д4, ленточного конвеера ЛК5, "куста" №1, "куста" №2 и разрешение на пуск следующей ступени агрегатов *)
work_level_61 := work_D4 AND work_LK5 AND work_level_2 AND work_level_4;
(* Network 42: Проверка готовности ленточных питателей ЛП4 и ЛП5. После пуска всех агрегатов этой ступени, / промежуточное реле самоподхвата разрывается для защиты от повторного пуска *)
prom7 := (pusk AND ready_LP4 AND (ready_LP5 OR in_040) OR prom7 AND NOT work_LP4 AND NOT work_LP5) AND NOT STOP_SYS AND NOT stop_LAN_LP4_out AND NOT stop_LAN_LP5_out;
(* Network 43: Блок управления ленточного питателя ЛП4 *)
LP4(pusk := work_LK5 AND avto_all AND prom7, avto := avto_LP4, KU := KU_LP4, TZ := TZ_LP4, MD3 := MD2_LP4, P := P_LP4, stop_lv := work_level_6, GRIB := gribok, stop_s := stop_all, ruchnoe := ruchnoe_all, pusk_LAN := pusk_LAN_LP4_out, stop_LAN := stop_LAN_LP4_out, err := e_LP4_out);
ready_LP4 := LP4.ready;
work_LP4 := LP4.work;
avar_LP4 := LP4.avar;
metall_LP4 := LP4.metall_LK4;
KM1_LP4 := LP4.KM;
(* Network 44: Блок управления ленточного питателя ЛП5 *)
LP5(pusk := work_LK5 AND avto_all AND prom7, avto := avto_LP5, STOP := STOP_LP5, VL := TRUE, MD2 := MD2_LP5, stop_lv := work_level_61, GRIB := gribok, input_Hz := out_Hz_LP5, stop_s := stop_all, pusk_LAN := pusk_LAN_LP5_out, stop_LAN := stop_LAN_LP5_out, P := in_P_LP5, ruchnoe := ruchnoe_all, ins_0_40 := in_040, err := e_LP5_out, pusk_sys_ins := PUSK_SYS, avar_FC := avar_FC_LP5);
pusk_LP5 := LP5.KM;
work_LP5 := LP5.work;
avar_LP5 := LP5.avar;
metall_LP5 := LP5.met;
b1_00_LP5 := LP5.b1_00;
b1_04_LP5 := LP5.b1_04;
avto_out_LP5 := LP5.avto_in;
avar_vl_lp5 := LP5.avar_vl;
ready_LP5 := LP5.ready;
(* Network 45 *)
stop_vl_lv3 := avar_vl_lk5 OR stop_vl_lv2;
(* Network 46: Проверка готовности ленточного конвеера ЛК4. После пуска всех агрегатов этой ступени, / промежуточное реле самоподхвата разрывается для защиты от повторного пуска *)
prom8 := (pusk AND ready_LK4 OR prom8 AND NOT avar_LK4 AND NOT work_LK4) AND NOT STOP_SYS AND NOT stop_lan_LK4_out;
(* Network 47: Блок управления ленточного конвеера ЛК4 *)
ton_LK4(IN := work_LK5, PT := t#1s);
LK4(pusk := ton_LK4.Q AND avto_all AND prom8, avto := avto_LK4, KU := KU_LK4, TZ := TZ_LK4, tros := tros_LK4, shod := shod_LK4, MD3 := MD3_LK4, VL := bool_Vl_LK4, P := P_LK4, stop_lv := work_D2 AND work_level_4 AND work_lk5 AND work_level_2, GRIB := gribok, stop_s := stop_all, ruchnoe := ruchnoe_all, pusk_LAN := pusk_lan_LK4_out, stop_LAN := stop_lan_LK4_out, err := e_LK4_out, tros_self := tros_self_lk4_out, shod_self := shod_self_lk4_out, pusk_sys_ins := PUSK_SYS);
ready_LK4 := LK4.ready;
work_LK4 := LK4.work;
avar_LK4 := LK4.avar;
metall_LK4 := LK4.metall_LK4;
avar_vl_lk4 := LK4.avar_vl;
KM1_LK4 := LK4.KM;
(* Network 48 *)
prom10 := (pusk AND ready_VP1 OR prom10 AND NOT work_VP1 AND NOT avar_VP1) AND NOT STOP_SYS AND NOT stop_LAN_VP1_out;
(* Network 49: Блок управления вибропитателя ВП1 *)
VP1(pusk := work_LK4 AND avto_all AND prom10, avto := avto_VP1, KU := KU_VP1, TZ := TZ_VP1, STOP := STOP_VP1, stop_lv := work_LK4, GRIB := gribok, LV_low_LK7 := TRUE, LV_high_LK7 := FALSE, LV_low_LK8 := TRUE, LV_high_LK8 := FALSE, LV_low_D2 := LV_low_D2, LV_high_D2 := LV_high_D2, stop_s := stop_all, pusk_LAN := pusk_LAN_VP1_out, stop_LAN := stop_LAN_VP1_out, P := P_VP1, err := e_VP1_out OR e_lp4_temp_out);
pusk_VP1 := VP1.KM;
work_VP1 := VP1.work;
avar_VP1 := VP1.avar;
ready_VP1 := VP1.ready;
(* Network 50: Проверка готовности ленточного конвеера ЛК2, ЛК3, грохота ГР1 и вибропитателя ВП1. После пуска всех агрегатов этой ступени, / промежуточное реле самоподхвата разрывается для защиты от повторного пуска *)
prom9 := (pusk AND ready_GR1 AND ready_LK2 AND ready_LK3 OR prom9 AND NOT work_level_9 AND NOT avar_LK3 AND NOT avar_LK2 AND NOT avar_VP1) AND NOT STOP_SYS AND NOT stop_lan_LK3_out AND NOT stop_lan_GR1_out AND NOT stop_lan_LK2_out;
(* Network 51: Блок управления ленточного конвеера ЛК3 *)
ton_LK3(IN := work_LK4, PT := t#1s);
LK3(pusk := ton_LK3.Q AND avto_all AND prom9, avto := avto_LK3, KU := KU_LK3, TZ := TZ_LK3, tros := tros_LK3, shod := shod_LK3, ogr := ogr_LK3, VL := bool_Vl_LK3, P := P_LK3, GRIB := stop_all, stop_s := gribok, ruchnoe := ruchnoe_all, pusk_LAN := pusk_lan_LK3_out, stop_LAN := stop_lan_LK3_out, err := e_LK3_out, tros_self := tros_self_lk3_out, shod_self := shod_self_lk3_out, ogr_self := ogr_self_lk3_out, pusk_sys_ins := PUSK_SYS);
ready_LK3 := LK3.ready;
work_LK3 := LK3.work;
avar_LK3 := LK3.avar;
avar_vl_lk3 := LK3.avar_vl;
KM1_LK3 := LK3.KM;
(* Network 52: Блок управления грохота ГР1 *)
ton_GR1(IN := work_LK3, PT := t#1s);
GR1(pusk := ton_GR1.Q AND avto_all AND prom9, avto := avto_GR1, KU := KU_GR1, TZ := TZ_GR1, P := P_GR1, STOP := STOP_GR1, GRIB := stop_all, stop_s := gribok, ruchnoe := ruchnoe_all, pusk_LAN := pusk_lan_GR1_out, stop_LAN := stop_lan_GR1_out, err := e_GR1_out);
ready_GR1 := GR1.ready;
work_GR1 := GR1.work;
avar_GR1 := GR1.avar;
KM1_GR1 := GR1.KM;
(* Network 53: Блок управления ленточного конвеера ЛК2 *)
ton_LK2(IN := work_GR1, PT := t#10s);
LK2(pusk := ton_LK2.Q AND avto_all AND prom9, avto := avto_LK2, KU := KU_LK2, TZ := TZ_LK2, tros := tros_LK2, shod := shod_LK2, ogr := ogr_LK2, VL := bool_Vl_LK2, P := P_LK2, GRIB := gribok, stop_s := stop_all, stop_lv := work_GR1, ruchnoe := ruchnoe_all, pusk_LAN := pusk_lan_LK2_out, stop_LAN := stop_lan_LK2_out, err := e_LK2_out, tros_self := tros_self_lk2_out, shod_self := shod_self_lk2_out, ogr_self := ogr_self_lk2_out, pusk_sys_ins := PUSK_SYS);
ready_LK2 := LK2.ready;
work_LK2 := LK2.work;
avar_LK2 := LK2.avar;
avar_vl_lk2 := LK2.avar_vl;
KM1_LK2 := LK2.KM;
(* Network 54: Подтверждение работы ленточных конвееров ЛК2, ЛК3, грохота ГР1 и вибропитателя ВП1 *)
work_level_9 := work_LK2 AND work_LK3 AND work_GR1;
(* Network 55: Блок отключения пластинчатого питателя ПП1 *)
PP1_blok(P_LK2_in := work_LK2, stop_pp_LK3 := work_LK3, LV2 := LV_low_GR1, LV1 := LV_high_GR1, pusk_s := pusk_sys, stop_s := stop_sys);
PP1 := PP1_blok.KM1_PP1;
(* Network 56: Блок управления битовой маской выходов модуля расширения в шкафу управления ЛК2 *)
LK2_out := PACK(KM1_LK2, FALSE, PP1, FALSE, FALSE, FALSE, FALSE, FALSE);
(* Network 57: Блоки управления отключением вибропитателя ВП1, ленточных конвееров ЛК7 и ЛК8 в зависимости от уровня в бункере *)
stop_VP1_LK7(LV_in := 4-LV_LK7, LV_high_in := ust_LV2_LK7, LV_low_in := ust_LV1_LK7);
LV_low_LK7 := stop_VP1_LK7.LV1_out;
LV_high_LK7 := stop_VP1_LK7.LV2_out;
stop_VP1_LK8(LV_in := 4-LV_LK8, LV_high_in := ust_LV2_LK8, LV_low_in := ust_LV1_LK8);
LV_low_LK8 := stop_VP1_LK8.LV1_out;
LV_high_LK8 := stop_VP1_LK8.LV2_out;
stop_VP1_D2(LV_in := 2.2-LV_D2, LV_high_in := ust_LV2_D2, LV_low_in := ust_LV1_D2);
LV_low_D2 := stop_VP1_D2.LV1_out;
LV_high_D2 := stop_VP1_D2.LV2_out;
stop_PP1(LV_in := LV_GR1 - 0.8, LV_high_in := ust_LV2_GR1, LV_low_in := ust_LV1_GR1);
LV_low_GR1 := stop_PP1.LV1_out;
LV_high_GR1 := stop_PP1.LV2_out;
if_Hz(input_Hz_LP4_if := input_Hz_LP4, input_Hz_LP5_if := input_Hz_LP5);
out_Hz_LP5 := if_Hz.output_Hz_LP5_if;
out_Hz_LP4 := if_Hz.output_Hz_LP4_if;
if_LV(input_LV2_LK7 := ust_LV2_LK7, input_LV1_LK7 := ust_LV1_LK7, input_LV2_LK8 := ust_LV2_LK8, input_LV1_LK8 := ust_LV1_LK8, input_LV2_GR1 := ust_LV2_GR1, input_LV1_GR1 := ust_LV1_GR1, input_LV2_D2 := ust_LV2_D2, input_LV1_D2 := ust_LV1_D2, input_time_VL := time_VL);
ust_LV1_LK7 := if_LV.output_LV1_LK7;
ust_LV2_LK8 := if_LV.output_LV2_LK8;
ust_LV1_LK8 := if_LV.output_LV1_LK8;
ust_LV2_GR1 := if_LV.output_LV2_GR1;
ust_LV1_GR1 := if_LV.output_LV1_GR1;
ust_LV2_D2 := if_LV.output_LV2_D2;
ust_LV1_D2 := if_LV.output_LV1_D2;
time_VL := if_LV.output_time_VL;
ust_LV2_LK7 := if_LV.output_LV2_LK7;
(* Network 58: Вывод аварии, в виде световой сигнализации, на шкаф контроллера *)
avaria := avar_D3 OR avar_D4 OR avar_LK10 OR avar_LK11 OR avar_LK12 OR avar_LK13 OR avar_GR3 OR avar_LK7 OR avar_LK6 OR avar_LK9 OR avar_LP1_3 OR avar_GR2 OR avar_LK5 OR avar_LP4 OR avar_LP5 OR avar_GR1 OR avar_LK4 OR avar_Lk2 OR avar_VP1 OR avar_LK3 OR gribok;
(* Network 59: Вывод наличия, в виде световой сигнализации, на шкаф контроллера *)
metall := metall_LP4 OR metall_LP5 OR metall_LK4;
(* Network 60: Блоки управления подсчетом скорости вращения *)
counter_LK10(Vl := Vl_LK10, work := work_lk10, in_time := time_VL);
bool_Vl_LK10 := counter_LK10.out_Vl;
counter_LK11(Vl := Vl_LK11, work := work_lk11, in_time := time_VL);
bool_Vl_LK11 := counter_LK11.out_Vl;
counter_LK12(Vl := Vl_LK12, work := work_lk12, in_time := time_VL);
bool_Vl_LK12 := counter_LK12.out_Vl;
counter_LK13(Vl := Vl_LK13, work := work_lk13, in_time := time_VL);
bool_Vl_LK13 := counter_LK13.out_Vl;
counter_LK7(Vl := Vl_LK7, work := work_lk7, in_time := time_VL);
bool_Vl_LK7 := counter_LK7.out_Vl;
counter_LK8(Vl := Vl_LK8, work := work_lk8, in_time := time_VL);
bool_Vl_LK8 := counter_LK8.out_Vl;
counter_LK6(Vl := Vl_LK6, work := work_lk6, in_time := time_VL);
bool_Vl_LK6 := counter_LK6.out_Vl;
counter_LK9(Vl := Vl_LK9, work := work_lk9, in_time := time_VL);
bool_Vl_LK9 := counter_LK9.out_Vl;
counter_LP1_3_1(Vl := Vl1_LP1_3, work := work_LP1_3, in_time := time_VL);
bool_Vl1_LP1_3 := counter_LP1_3_1.out_Vl;
counter_LP1_3_2(Vl := Vl2_LP1_3, work := work_LP1_3, in_time := time_VL);
bool_Vl2_LP1_3 := counter_LP1_3_2.out_Vl;
counter_LP1_3_3(Vl := Vl3_LP1_3, work := work_LP1_3, in_time := time_VL);
bool_Vl3_LP1_3 := counter_LP1_3_3.out_Vl;
counter_LK5(Vl := Vl_LK5, work := work_lk5, in_time := time_VL);
bool_Vl_LK5 := counter_LK5.out_Vl;
counter_LP5(Vl := Vl_LP5, work := work_lp5, in_time := time_VL);
bool_Vl_LP5 := counter_LP5.out_Vl;
counter_LK4(Vl := Vl_LK4, work := work_lk4, in_time := time_VL);
bool_Vl_LK4 := counter_LK4.out_Vl;
counter_LK3(Vl := Vl_LK3, work := work_lk3, in_time := time_VL);
bool_Vl_LK3 := counter_LK3.out_Vl;
counter_LK2(Vl := Vl_LK2, work := work_lk2, in_time := time_VL);
bool_Vl_LK2 := counter_LK2.out_Vl;
(* Network 61: Блок вывода сигналов для SCADA-системы *)
signals(KU_D2_in := KU_D2, RMS2_2_in := RMS2_2, avto_D2_in := avto_D2, work_D2_in := work_D2, ready_D2_in := ready_D2, TZD2_in := TZD2, KU_D3_in := KU_D3, TZN_D3_in := TZN_D3, UM_D3_in := UM_D3, KPM_D3_in := KPM_D3, TZV_D3_in := TZV_D3, avto_D3_in := avto_D3, KUD3_D3_in := KUD3_D3, TZD3_D3_in := TZD3_D3, work_D3_in := work_D3, ready_D3_in := ready_D3, TM_D3_in := TM_D3_bool, RMS_D3_in := RMS_D3, DM_D3_in := DM_D3, KU_D4_in := KU_D4, TZN_D4_in := TZN_D4, UM_D4_in := UM_D4, KPM_D4_in := KPM_D4, TZV_D4_in := TZV_D4, avto_D4_in := avto_D4, KUD3_D4_in := KUD3_D4, TZD3_D4_in := TZD3_D4, work_D4_in := work_D4, ready_D4_in := ready_D4, TM_D4_in := TM_D4_bool, RMS_D4_in := RMS_D4, DM_D4_in := DM_D4, KU_LK10_in := KU_LK10, TZ_LK10_in := TZ_LK10, tros_LK10_in := tros_LK10, shod_LK10_in := shod_LK10, ogr_LK10_in := ogr_LK10, avto_LK10_in := avto_LK10, ready_LK10_in := ready_LK10, work_LK10_in := work_LK10, KU_LK11_in := KU_LK11, TZ_LK11_in := TZ_LK11, tros_LK11_in := tros_LK11, shod_LK11_in := shod_LK11, ogr_LK11_in := ogr_LK11, avto_LK11_in := avto_LK11, ready_LK11_in := ready_LK11, work_LK11_in := work_LK11, KU_LK12_in := KU_LK12, TZ_LK12_in := TZ_LK12, tros_LK12_in := tros_LK12, shod_LK12_in := shod_LK12, ogr_LK12_in := ogr_LK12, avto_LK12_in := avto_LK12, ready_LK12_in := ready_LK12, work_LK12_in := work_LK12, KU_LK13_in := KU_LK13, TZ_LK13_in := TZ_LK13, tros_LK13_in := tros_LK13, shod_LK13_in := shod_LK13, ogr_LK13_in := ogr_LK13, avto_LK13_in := avto_LK13, ready_LK13_in := ready_LK13, work_LK13_in := work_LK13, avto_GR3_in := avto_GR3, KU_GR3_in := KU_GR3, TZ_GR3_in := TZ_GR3, ready_GR3_in := ready_GR3, work_GR3_in := work_GR3, STOP_GR3_in := STOP_GR3, KU_LK7_in := KU_LK7, TZ_LK7_in := TZ_LK7, tros_LK7_in := tros_LK7, shod_LK7_in := shod_LK7, ogr_LK7_in := ogr_LK7, avto_LK7_in := avto_LK7, ready_LK7_in := ready_LK7, work_LK7_in := work_LK7, KU_LK8_in := KU_LK8, TZ_LK8_in := TZ_LK8, tros_LK8_in := tros_LK8, shod_LK8_in := shod_LK8, ogr_LK8_in := ogr_LK8, avto_LK8_in := avto_LK8, ready_LK8_in := ready_LK8, work_LK8_in := work_LK8, KU_LK6_in := KU_LK6, TZ_LK6_in := TZ_LK6, tros_LK6_in := tros_LK6, shod_LK6_in := shod_LK6, ogr_LK6_in := ogr_LK6, avto_LK6_in := avto_LK6, ready_LK6_in := ready_LK6, work_LK6_in := work_LK6, KU_LK9_in := KU_LK9, TZ_LK9_in := TZ_LK9, tros_LK9_in := tros_LK9, ogr_LK9_in := ogr_LK9, shod_LK9_in := shod_LK9, avto_LK9_in := avto_LK9, ready_LK9_in := ready_LK9, work_LK9_in := work_LK9, KU_LP1_3_in := KU_LP1_3, in_020_in := in_020, in_040_in := in_040, in_020_4070_in := in_020_4070, TZ1_LP1_3_in := TZ1_LP1_3, TZ2_LP1_3_in := TZ2_LP1_3, TZ3_LP1_3_in := TZ3_LP1_3, PRO_LP1_3_in := PRO_LP1_3, avto_LP1_3_in := avto_LP1_3, ready_LP1_3_in := ready_LP1_3, work_LP1_3_in := work_LP1_3, stop2_LP1_3_in := stop2_LP1_3, avto_GR2_in := avto_GR2, KU_GR2_in := KU_GR2, TZ_GR2_in := TZ_GR2, ready_GR2_in := ready_GR2, work_GR2_in := work_GR2, STOP_GR2_in := STOP_GR2, KU_LK5_in := KU_LK5, TZ_LK5_in := TZ_LK5, tros_LK5_in := tros_LK5, shod_LK5_in := shod_LK5, ogr_LK5_in := ogr_LK5, avto_LK5_in := avto_LK5, ready_LK5_in := ready_LK5, work_LK5_in := work_LK5, KU_LK4_in := KU_LK4, TZ_LK4_in := TZ_LK4, tros_LK4_in := tros_LK4, shod_LK4_in := shod_LK4, avto_LK4_in := avto_LK4, ready_LK4_in := ready_LK4, work_LK4_in := work_LK4, MD3_LK4_in := metall_LK4, avto_GR1_in := avto_GR1, KU_GR1_in := KU_GR1, TZ_GR1_in := TZ_GR1, ready_GR1_in := ready_GR1, work_GR1_in := work_GR1, STOP_GR1_in := STOP_GR1, KU_LK2_in := KU_LK2, TZ_LK2_in := TZ_LK2, tros_LK2_in := tros_LK2, shod_LK2_in := shod_LK2, ogr_LK2_in := ogr_LK2, avto_LK2_in := avto_LK2, ready_LK2_in := ready_LK2, work_LK2_in := work_LK2, KU_LK3_in := KU_LK3, TZ_LK3_in := TZ_LK3, tros_LK3_in := tros_LK3, shod_LK3_in := shod_LK3, ogr_LK3_in := ogr_LK3, avto_LK3_in := avto_LK3, ready_LK3_in := ready_LK3, work_LK3_in := work_LK3, avto_LP4_in := avto_LP4, ready_LP4_in := ready_LP4, work_LP4_in := work_LP4, MD2_LP4_in := metall_LP4, avto_LP5_in := avto_LP5, ready_LP5_in := ready_LP5, work_LP5_in := work_LP5, STOP_LP5_in := STOP_LP5, output_Hz_LP5_in := output_Hz_LP5, MD2_LP5_in := metall_LP5, avto_VP1_in := avto_VP1, ready_VP1_in := ready_VP1, work_VP1_in := work_VP1, STOP_VP1_in := STOP_VP1, KU_VP1_in := KU_VP1, TZ_VP1_in := TZ_VP1, avto_all_in := avto_all, pusk_in := pusk_lan, PP1_in := PP1, LV_GR1_in := LV_GR1, LV_LK7_in := LV_LK7, LV_LK8_in := LV_LK8, LV_D2_in := LV_D2, lev_up_cyc_in := lev_up_cyc, pre_cyc_in := pre_cyc, ku_cyc_in := ku_cyc, tz_cyc_in := tz_cyc, ready_cyc_in := ready_cyc, work_cyc_in := work_cyc, shnek_up_cyc_in := shnek_up_cyc, avar_cyc_in := avar_cyc, gribok_in := gribok, TM_D3_word_in := TM_D3, TM_D4_word_in := TM_D4, avar_FC_lp5_in := avar_FC_LP5, lev_down_cyc_in := lev_down_cyc);
RMS_2_2_out := signals.RMS2_2_out;
avto_D2_out := signals.avto_D2_out;
work_D2_out := signals.work_D2_out;
ready_D2_out := signals.ready_D2_out;
TZD2_out := signals.TZD2_out;
KU_D3_out := signals.KU_D3_out;
TZN_D3_out := signals.TZN_D3_out;
UM_D3_out := signals.UM_D3_out;
KPM_D3_out := signals.KPM_D3_out;
TZV_D3_out := signals.TZV_D3_out;
avto_D3_out := signals.avto_D3_out;
KUD3_D3_out := signals.KUD3_D3_out;
TZD3_D3_out := signals.TZD3_D3_out;
work_D3_out := signals.work_D3_out;
ready_D3_out := signals.ready_D3_out;
TM_D3_out := signals.TM_D3_out;
RMS_D3_out := signals.RMS_D3_out;
DM_D3_out := signals.DM_D3_out;
KU_D4_out := signals.KU_D4_out;
TZN_D4_out := signals.TZN_D4_out;
UM_D4_out := signals.UM_D4_out;
KPM_D4_out := signals.KPM_D4_out;
TZV_D4_out := signals.TZV_D4_out;
KUD3_D4_out := signals.KUD3_D4_out;
TZD3_D4_out := signals.TZD3_D4_out;
work_D4_out := signals.work_D4_out;
ready_D4_out := signals.ready_D4_out;
avto_D4_out := signals.avto_D4_out;
TM_D4_out := signals.TM_D4_out;
RMS_D4_out := signals.RMS_D4_out;
DM_D4_out := signals.DM_D4_out;
KU_LK10_out := signals.KU_LK10_out;
TZ_LK10_out := signals.TZ_LK10_out;
tros_LK10_out := signals.tros_LK10_out;
shod_LK10_out := signals.shod_LK10_out;
ogr_LK10_out := signals.ogr_LK10_out;
avto_LK10_out := signals.avto_LK10_out;
ready_LK10_out := signals.ready_LK10_out;
work_LK10_out := signals.work_LK10_out;
KU_LK11_out := signals.KU_LK11_out;
TZ_LK11_out := signals.TZ_LK11_out;
tros_LK11_out := signals.tros_LK11_out;
shod_LK11_out := signals.shod_LK11_out;
ogr_LK11_out := signals.ogr_LK11_out;
ato_LK11_out := signals.avto_LK11_out;
ready_LK11_out := signals.ready_LK11_out;
work_LK11_out := signals.work_LK11_out;
KU_LK12_out := signals.KU_LK12_out;
TZ_LK12_out := signals.TZ_LK12_out;
tros_LK12_out := signals.tros_LK12_out;
shod_LK12_out := signals.shod_LK12_out;
ogr_LK12_out := signals.ogr_LK12_out;
avto_LK12_out := signals.avto_LK12_out;
ready_LK12_out := signals.ready_LK12_out;
work_LK12_out := signals.work_LK12_out;
KU_LK13_out := signals.KU_LK13_out;
TZ_LK13_out := signals.TZ_LK13_out;
tros_LK13_out := signals.tros_LK13_out;
shod_LK13_out := signals.shod_LK13_out;
ogr_LK13_out := signals.ogr_LK13_out;
avto_LK13_out := signals.avto_LK13_out;
ready_LK13_out := signals.ready_LK13_out;
work_LK13_out := signals.work_LK13_out;
avto_GR3_out := signals.avto_GR3_out;
KU_GR3_out := signals.KU_GR3_out;
TZ_GR3_out := signals.TZ_GR3_out;
ready_GR3_out := signals.ready_GR3_out;
work_GR3_out := signals.work_GR3_out;
STOP_GR3_out := signals.STOP_GR3_out;
KU_LK7_out := signals.KU_LK7_out;
TZ_LK7_out := signals.TZ_LK7_out;
tros_LK7_out := signals.tros_LK7_out;
shod_LK7_out := signals.shod_LK7_out;
ogr_LK7_out := signals.ogr_LK7_out;
avto_LK7_out := signals.avto_LK7_out;
ready_LK7_out := signals.ready_LK7_out;
work_LK7_out := signals.work_LK7_out;
KU_LK8_out := signals.KU_LK8_out;
TZ_LK8_out := signals.TZ_LK8_out;
tros_LK8_out := signals.tros_LK8_out;
shod_LK8_out := signals.shod_LK8_out;
ogr_LK8_out := signals.ogr_LK8_out;
avto_LK8_out := signals.avto_LK8_out;
ready_LK8_out := signals.ready_LK8_out;
work_LK8_out := signals.work_LK8_out;
KU_LK6_out := signals.KU_LK6_out;
TZ_LK6_out := signals.TZ_LK6_out;
tros_LK6_out := signals.tros_LK6_out;
shod_LK6_out := signals.shod_LK6_out;
ogr_LK6_out := signals.ogr_LK6_out;
avto_LK6_out := signals.avto_LK6_out;
ready_LK6_out := signals.ready_LK6_out;
work_LK6_out := signals.work_LK6_out;
KU_LK9_out := signals.KU_LK9_out;
TZ_LK9_out := signals.TZ_LK9_out;
tros_LK9_out := signals.tros_LK9_out;
shod_LK9_out := signals.shod_LK9_out;
ogr_LK9_out := signals.ogr_LK9_out;
avto_LK9_out := signals.avto_LK9_out;
ready_LK9_out := signals.ready_LK9_out;
work_LK9_out := signals.work_LK9_out;
KU_LP1_3_out := signals.KU_LP1_3_out;
in_020_out := signals.in_020_out;
in_040_out := signals.in_040_out;
in_020_4070_out := signals.in_020_4070_out;
TZ1_LP1_3_out := signals.TZ1_LP1_3_out;
TZ2_LP1_3_out := signals.TZ2_LP1_3_out;
TZ3_LP1_3_out := signals.TZ3_LP1_3_out;
PRO_LP1_3_out := signals.PRO_LP1_3_out;
avto_LP1_3_out := signals.avto_LP1_3_out;
ready_LP1_3_out := signals.ready_LP1_3_out;
work_LP1_3_out := signals.work_LP1_3_out;
stop2_LP1_3_out := signals.stop2_LP1_3_out;
avto_GR2_out := signals.avto_GR2_out;
KU_GR2_out := signals.KU_GR2_out;
TZ_GR2_out := signals.TZ_GR2_out;
ready_GR2_out := signals.ready_GR2_out;
work_GR2_out := signals.work_GR2_out;
STOP_GR2_out := signals.STOP_GR2_out;
KU_LK5_out := signals.KU_LK5_out;
TZ_LK5_out := signals.TZ_LK5_out;
tros_LK5_out := signals.tros_LK5_out;
shod_LK5_out := signals.shod_LK5_out;
ogr_LK5_out := signals.ogr_LK5_out;
avto_LK5_out := signals.avto_LK5_out;
ready_LK5_out := signals.ready_LK5_out;
work_LK5_out := signals.work_LK5_out;
KU_LK4_out := signals.KU_LK4_out;
TZ_LK4_out := signals.TZ_LK4_out;
tros_LK4_out := signals.tros_LK4_out;
shod_LK4_out := signals.shod_LK4_out;
avto_LK4_out := signals.avto_LK4_out;
ready_LK4_out := signals.ready_LK4_out;
work_LK4_out := signals.work_LK4_out;
MD3_LK4_out := signals.MD3_LK4_out;
avto_GR1_out := signals.avto_GR1_out;
KU_GR1_out := signals.KU_GR1_out;
TZ_GR1_out := signals.TZ_GR1_out;
ready_GR1_out := signals.ready_GR1_out;
work_GR1_out := signals.work_GR1_out;
STOP_GR1_out := signals.STOP_GR1_out;
KU_LK2_out := signals.KU_LK2_out;
TZ_LK2_out := signals.TZ_LK2_out;
tros_LK2_out := signals.tros_LK2_out;
shod_LK2_out := signals.shod_LK2_out;
ogr_LK2_out := signals.ogr_LK2_out;
avto_LK2_out := signals.avto_LK2_out;
ready_LK2_out := signals.ready_LK2_out;
work_LK2_out := signals.work_LK2_out;
KU_LK3_out := signals.KU_LK3_out;
TZ_LK3_out := signals.TZ_LK3_out;
tros_LK3_out := signals.tros_LK3_out;
shod_LK3_out := signals.shod_LK3_out;
ogr_LK3_out := signals.ogr_LK3_out;
avto_LK3_out := signals.avto_LK3_out;
ready_LK3_out := signals.ready_LK3_out;
work_LK3_out := signals.work_LK3_out;
avto_LP4_out := signals.avto_LP4_out;
ready_LP4_out := signals.ready_LP4_out;
work_LP4_out := signals.work_LP4_out;
MD2_LP4_out := signals.MD2_LP4_out;
output_Hz_LP4_out := signals.output_Hz_LP4_out;
avto_LP5_out := signals.avto_LP5_out;
ready_LP5_out := signals.ready_LP5_out;
work_LP5_out := signals.work_LP5_out;
STOP_LP5_out := signals.STOP_LP5_out;
MD2_LP5_out := signals.MD2_LP5_out;
output_Hz_LP5_out := signals.output_Hz_LP5_out;
avto_VP1_out := signals.avto_VP1_out;
ready_VP1_out := signals.ready_VP1_out;
work_VP1_out := signals.work_VP1_out;
STOP_VP1_out := signals.STOP_VP1_out;
KU_VP1_out := signals.KU_VP1_out;
TZ_VP1_out := signals.TZ_VP1_out;
avto_all_out := signals.avto_all_out;
pusk_out := signals.pusk_out;
PP1_out := signals.PP1_out;
LV_GR1_out := signals.LV_GR1_out;
LV_LK7_out := signals.LV_LK7_out;
LV_LK8_out := signals.LV_LK8_out;
LV_D2_out := signals.LV_D2_out;
lev_up_cyc_out := signals.lev_up_cyc_out;
pre_cyc_out := signals.pre_cyc_out;
ku_cyc_out := signals.ku_cyc_out;
tz_cyc_out := signals.tz_cyc_out;
ready_cyc_out := signals.ready_cyc_out;
work_cyc_out := signals.work_cyc_out;
shnek_up_cyc_out := signals.shnek_up_cyc_out;
avar_cyc_out := signals.avar_cyc_out;
gribok_out := signals.gribok_out;
TM_D3_word_out := signals.TM_D3_word_out;
TM_D4_word_out := signals.TM_D4_word_out;
avar_FC_LP5_out := signals.avar_FC_lp5_out;
lev_down_cyc_out := signals.lev_down_cyc_out;
KU_D2_out := signals.KU_D2_out;
(* Network 62 *)
signals1(pusk_LAN_LP4 := pusk_LAN_LP4, stop_LAN_LP4 := stop_LAN_LP4, pusk_LAN_LP5 := pusk_LAN_LP5, stop_LAN_LP5 := stop_LAN_LP5, pusk_LAN_VP1 := pusk_LAN_VP1, stop_LAN_VP1 := stop_LAN_VP1, pusk_lan_LK10 := pusk_lan_LK10, pusk_lan_LK11 := pusk_lan_LK11, pusk_lan_LK12 := pusk_lan_LK12, pusk_lan_LK13 := pusk_lan_LK13, pusk_lan_GR3 := pusk_lan_GR3, pusk_lan_LK7 := pusk_lan_LK7, pusk_lan_LK8 := pusk_lan_LK8, pusk_lan_LK6 := pusk_lan_LK6, pusk_lan_LK9 := pusk_lan_LK9, pusk_lan_LP1_3 := pusk_lan_LP1_3, pusk_lan_GR2 := pusk_lan_GR2, pusk_lan_LK5 := pusk_lan_LK5, pusk_lan_LK4 := pusk_lan_LK4, pusk_lan_LK3 := pusk_lan_LK3, pusk_lan_GR1 := pusk_lan_GR1, pusk_lan_LK2 := pusk_lan_LK2, stop_lan_LK10 := stop_lan_LK10, stop_lan_LK11 := stop_lan_LK11, stop_lan_LK12 := stop_lan_LK12, stop_lan_LK13 := stop_lan_LK13, stop_lan_GR3 := stop_lan_GR3, stop_lan_LK7 := stop_lan_LK7, stop_lan_LK8 := stop_lan_LK8, stop_lan_LK6 := stop_lan_LK6, stop_lan_LK9 := stop_lan_LK9, stop_lan_LP1_3 := stop_lan_LP1_3, stop_lan_GR2 := stop_lan_GR2, stop_lan_LK5 := stop_lan_LK5, stop_lan_LK4 := stop_lan_LK4, stop_lan_LK3 := stop_lan_LK3, stop_lan_GR1 := stop_lan_GR1, stop_lan_LK2 := stop_lan_LK2, stop_LAN_D3 := stop_LAN_D3, stop_LAN_D4 := stop_LAN_D4, pusk_lan_D2 := pusk_LAN_D2, stop_lan_D2 := stop_LAN_D2, pusk_lan_D3 := pusk_LAN_D3, pusk_lan_D4 := pusk_LAN_D4, pusk_lan_cyclone := pusk_lan_cyclone, stop_lan_cyclone := stop_lan_cyclone, tros_self_lk10_in := tros_self_lk10, shod_self_lk10_in := shod_self_lk10, ogr_self_lk10_in := ogr_self_lk10, vl_self_lk10_in := vl_self_lk10, tros_self_lk11_in := tros_self_lk11, shod_self_lk11_in := shod_self_lk11, ogr_self_lk11_in := ogr_self_lk11, vl_self_lk11_in := vl_self_lk11, tros_self_lk12_in := tros_self_lk12, shod_self_lk12_in := shod_self_lk12, ogr_self_lk12_in := ogr_self_lk12, vl_self_lk12_in := vl_self_lk12, tros_self_lk13_in := tros_self_lk13, shod_self_lk13_in := shod_self_lk13, ogr_self_lk13_in := ogr_self_lk13, vl_self_lk13_in := vl_self_lk13, tros_self_lk7_in := tros_self_lk7, shod_self_lk7_in := shod_self_lk7, ogr_self_lk7_in := ogr_self_lk7, vl_self_lk7_in := vl_self_lk7, tros_self_lk8_in := tros_self_lk8, shod_self_lk8_in := shod_self_lk8, ogr_self_lk8_in := ogr_self_lk8, vl_self_lk8_in := vl_self_lk8, tros_self_lk6_in := tros_self_lk6, shod_self_lk6_in := shod_self_lk6, ogr_self_lk6_in := ogr_self_lk6, vl_self_lk6_in := vl_self_lk6, tros_self_lk9_in := tros_self_lk9, shod_self_lk9_in := shod_self_lk9, ogr_self_lk9_in := ogr_self_lk9, vl_self_lk9_in := vl_self_lk9, vl_self_lp1_3_in := vl_self_lp1_3, tros_self_lk5_in := tros_self_lk5, shod_self_lk5_in := shod_self_lk5, ogr_self_lk5_in := ogr_self_lk5, vl_self_lk5_in := vl_self_lk5, tros_self_lk4_in := tros_self_lk4, shod_self_lk4_in := shod_self_lk4, vl_self_lk4_in := vl_self_lk4, tros_self_lk3_in := tros_self_lk3, shod_self_lk3_in := shod_self_lk3, ogr_self_lk3_in := ogr_self_lk3, vl_self_lk3_in := vl_self_lk3, tros_self_lk2_in := tros_self_lk2, shod_self_lk2_in := shod_self_lk2, ogr_self_lk2_in := ogr_self_lk2, vl_self_lk2_in := vl_self_lk2, revers_in := revers, vl_self_lp4_in := vl_self_lp4, vl_self_lp5_in := vl_self_lp5, pusk_shnek_razg_in := pusk_shnek_razg, stop_shnek_razg_in := stop_shnek_razg, pusk_cyc_cleen_in := pusk_cleen_lan, stop_cyc_cleen_in := stop_cleen_lan);
stop_LAN_LP4_out := signals1.stop_LAN_LP4_out;
pusk_LAN_LP5_out := signals1.pusk_LAN_LP5_out;
stop_LAN_LP5_out := signals1.stop_LAN_LP5_out;
pusk_LAN_VP1_out := signals1.pusk_LAN_VP1_out;
stop_LAN_VP1_out := signals1.stop_LAN_VP1_out;
pusk_lan_LK10_out := signals1.pusk_lan_LK10_out;
pusk_lan_LK11_out := signals1.pusk_lan_LK11_out;
pusk_lan_LK12_out := signals1.pusk_lan_LK12_out;
pusk_lan_LK13_out := signals1.pusk_lan_LK13_out;
pusk_lan_GR3_out := signals1.pusk_lan_GR3_out;
pusk_lan_LK7_out := signals1.pusk_lan_LK7out;
pusk_lan_LK8_out := signals1.pusk_lan_LK8_out;
pusk_lan_LK6_out := signals1.pusk_lan_LK6_out;
pusk_lan_LK9_out := signals1.pusk_lan_LK9_out;
pusk_lan_LP1_3_out := signals1.pusk_lan_LP1_3_out;
pusk_lan_GR2_out := signals1.pusk_lan_GR2_out;
pusk_lan_LK5_out := signals1.pusk_lan_LK5_out;
pusk_lan_LK4_out := signals1.pusk_lan_LK4_out;
pusk_lan_LK3_out := signals1.pusk_lan_LK3_out;
pusk_lan_GR1_out := signals1.pusk_lan_GR1_out;
pusk_lan_LK2_out := signals1.pusk_lan_LK2_out;
stop_lan_LK10_out := signals1.stop_lan_LK10_out;
stop_lan_LK11_out := signals1.stop_lan_LK11_out;
stop_lan_LK12_out := signals1.stop_lan_LK12_out;
stop_lan_LK13_out := signals1.stop_lan_LK13_out;
stop_lan_GR3_out := signals1.stop_lan_GR3_out;
stop_lan_LK7_out := signals1.stop_lan_LK7_out;
stop_lan_LK8_out := signals1.stop_lan_LK8_out;
stop_lan_LK6_out := signals1.stop_lan_LK6_out;
stop_lan_LK9_out := signals1.stop_lan_LK9_out;
stop_lan_LP1_3_out := signals1.stop_lan_LP1_3_out;
stop_lan_GR2_out := signals1.stop_lan_GR2_out;
stop_lan_LK5_out := signals1.stop_lan_LK5_out;
stop_lan_LK4_out := signals1.stop_lan_LK4_out;
stop_lan_LK3_out := signals1.stop_lan_LK3_out;
stop_lan_GR1_out := signals1.stop_lan_GR1_out;
stop_lan_LK2_out := signals1.stop_lan_LK2_out;
stop_LAN_D3_out := signals1.stop_LAN_D3_out;
stop_LAN_D4_out := signals1.stop_LAN_D4_out;
pusk_LAN_D2_out := signals1.pusk_lan_D2_out;
stop_LAN_D2_out := signals1.stop_lan_D2_out;
pusk_LAN_D3_out := signals1.pusk_lan_D3_out;
pusk_LAN_D4_out := signals1.pusk_lan_D4_out;
pusk_lan_cyclone_out := signals1.pusk_lan_cyclone_out;
stop_lan_cyclone_out := signals1.stop_lan_cyclone_out;
tros_self_lk10_out := signals1.tros_self_lk10_out;
shod_self_lk10_out := signals1.shod_self_lk10_out;
ogr_self_lk10_out := signals1.ogr_self_lk10_out;
vl_self_lk10_out := signals1.vl_self_lk10_out;
tros_self_lk11_out := signals1.tros_self_lk11_out;
shod_self_lk11_out := signals1.shod_self_lk11_out;
ogr_self_lk11_out := signals1.ogr_self_lk11_out;
vl_self_lk11_out := signals1.vl_self_lk11_out;
tros_self_lk12_out := signals1.tros_self_lk12_out;
shod_self_lk12_out := signals1.shod_self_lk12_out;
ogr_self_lk12_out := signals1.ogr_self_lk12_out;
vl_self_lk12_out := signals1.vl_self_lk12_out;
tros_self_lk13_out := signals1.tros_self_lk13_out;
shod_self_lk13_out := signals1.shod_self_lk13_out;
ogr_self_lk13_out := signals1.ogr_self_lk13_out;
vl_self_lk13_out := signals1.vl_self_lk13_out;
tros_self_lk7_out := signals1.tros_self_lk7_out;
shod_self_lk7_out := signals1.shod_self_lk7_out;
ogr_self_lk7_out := signals1.ogr_self_lk7_out;
vl_self_lk7_out := signals1.vl_self_lk7_out;
tros_self_lk8_out := signals1.tros_self_lk8_out;
shod_self_lk8_out := signals1.shod_self_lk8_out;
ogr_self_lk8_out := signals1.ogr_self_lk8_out;
vl_self_lk8_out := signals1.vl_self_lk8_out;
tros_self_lk6_out := signals1.tros_self_lk6_out;
shod_self_lk6_out := signals1.shod_self_lk6_out;
ogr_self_lk6_out := signals1.ogr_self_lk6_out;
vl_self_lk6_out := signals1.vl_self_lk6_out;
tros_self_lk9_out := signals1.tros_self_lk9_out;
shod_self_lk9_out := signals1.shod_self_lk9_out;
ogr_self_lk9_out := signals1.ogr_self_lk9_out;
vl_self_lk9_out := signals1.vl_self_lk9_out;
vl_self_lp1_3_out := signals1.vl_self_lp1_3_out;
tros_self_lk5_out := signals1.tros_self_lk5_out;
shod_self_lk5_out := signals1.shod_self_lk5_out;
ogr_self_lk5_out := signals1.ogr_self_lk5_out;
vl_self_lk5_out := signals1.vl_self_lk5_out;
tros_self_lk4_out := signals1.tros_self_lk4_out;
shod_self_lk4_out := signals1.shod_self_lk4_out;
vl_self_lk4_out := signals1.vl_self_lk4_out;
tros_self_lk3_out := signals1.tros_self_lk3_out;
shod_self_lk3_out := signals1.shod_self_lk3_out;
ogr_self_lk3_out := signals1.ogr_self_lk3_out;
vl_self_lk3_out := signals1.vl_self_lk3_out;
tros_self_lk2_out := signals1.tros_self_lk2_out;
shod_self_lk2_out := signals1.shod_self_lk2_out;
ogr_self_lk2_out := signals1.ogr_self_lk2_out;
vl_self_lk2_out := signals1.vl_self_lk2_out;
revers_out := signals1.revers_out;
vl_self_lp4_out := signals1.vl_self_lp4_out;
vl_self_lp5_out := signals1.vl_self_lp5_out;
pusk_shnek_razg_out := signals1.pusk_shnek_razg_out;
stop_shnek_razg_out := signals1.stop_shnek_razg_out;
cyc_cleen_pusk := signals1.pusk_cyc_cleen_out;
cyc_cleen_stop := signals1.stop_cyc_cleen_out;
pusk_LAN_LP4_out := signals1.pusk_LAN_LP4_out;
(* Network 63 *)
alarm(adress_in_rs2 := adr_dev_rs2, error_81_in_rs2 := err_dev_rs2, adress_in_rs1 := adr_dev_rs1, error_81_in_rs1 := err_dev_rs1);
e_LK11_out := alarm.err_LK11;
e_LK12_out := alarm.err_LK12;
e_LK13_out := alarm.err_LK13;
e_GR3_out := alarm.err_GR3;
e_LK7_out := alarm.err_LK7;
e_LK8_out := alarm.err_LK8;
e_LK6_out := alarm.err_LK6;
e_LK9_out := alarm.err_LK9;
e_LP13mod1_out := alarm.err_LP1_3_mod1;
e_LP13mod2_out := alarm.err_LP1_3_mod2;
e_GR2_out := alarm.err_GR2;
e_LK5_out := alarm.err_LK5;
e_LP4_out := alarm.err_LP4;
e_LP5_out := alarm.err_LP5;
e_LK4_out := alarm.err_LK4;
e_GR1_out := alarm.err_GR1;
e_LK2_out := alarm.err_LK2;
e_LK3_out := alarm.err_LK3;
e_VP1_out := alarm.err_VP1;
e_D3mod1_out := alarm.err_D3_mod1;
e_D3mod2_out := alarm.err_D3_mod2;
e_D4mod1_out := alarm.err_D4_mod1;
e_D4mod2_out := alarm.err_D4_mod2;
e_D2_out := alarm.err_D2;
e_cyc1_out := alarm.err_cyc1;
e_cyc2_out := alarm.err_cyc2;
e_lp4_temp_out := alarm.err_lp4_temp;
e_d3_temp_out := alarm.err_d3_temp;
e_d4_temp_out := alarm.err_d4_temp;
e_vp1_temp_out := alarm.err_vp1_temp;
e_LK10_out := alarm.err_LK10;
alarm_all(err_LK10 := e_LK10_out, err_LK11 := e_LK11_out, err_LK12 := e_LK12_out, err_LK13 := e_LK13_out, err_GR3 := e_GR3_out, err_LK7 := e_LK7_out, err_LK8 := e_LK8_out, err_LK6 := e_LK6_out, err_LK9 := e_LK9_out, err_LP1_3_mod1 := e_LP13mod1_out, err_LP1_3_mod2 := e_LP13mod2_out, err_GR2 := e_GR2_out, err_LK5 := e_LK5_out, err_LP4 := e_LP4_out, err_LP5 := e_LP5_out, err_LK4 := e_LK4_out, err_GR1 := e_GR1_out, err_LK2 := e_LK2_out, err_LK3 := e_LK3_out, err_VP1 := e_VP1_out, err_D3_mod1 := e_D3mod1_out, err_D3_mod2 := e_D3mod2_out, err_D4_mod1 := e_D4mod1_out, err_D4_mod2 := e_D4mod2_out, err_D2 := e_D2_out, err_cyc1 := e_cyc1_out, err_cyc2 := e_cyc2_out, err_lp4_temp := e_lp4_temp_out, err_d3_temp := e_d3_temp_out, err_d4_temp := e_d4_temp_out, err_vp1_temp := e_vp1_temp_out);
moduls_out := alarm_all.modul_out;
END_PROGRAM

(* POU cyclone, LD *)
FUNCTION_BLOCK cyclone (*функциональный блок, управляющий работой элеватора (циклона)*)
VAR_INPUT
	stop: BOOL;
	grib: BOOL;
	pusk_LAN: BOOL;
	stop_lan: BOOL;
	level: BOOL;
	KU: BOOL;
	TZ: BOOL;
	skvaj: REAL;
	switch: BOOL;
	err: BOOL;
	pusk_shnek_lan: BOOL;
	stop_shnek_lan: BOOL;
	in_time: WORD;
	time_run: WORD;
	time_stop: WORD;
	cleen_in_pusk: BOOL;
	cleen_in_stop: BOOL;
END_VAR
VAR_OUTPUT
	vent: BOOL;
	VE_1: WORD;
	VE_2: WORD;
	VE_3: WORD;
	VE_4: WORD;
	VE_5: WORD;
	VE_6: WORD;
	VE_7: WORD;
	VE_8: WORD;
	shnek_up: BOOL;
	ready: BOOL;
	work: BOOL;
	avar: BOOL;
	shnek_razg: BOOL;
	prom_cleen_word: WORD;
END_VAR
VAR
	prom: BOOL;

	prom1: BOOL;
	prom2: BOOL;
	prom3: BOOL;
	prom4: BOOL;
	prom5: BOOL;
	prom6: BOOL;
	prom7: BOOL;
	prom8: BOOL;

	skv1: REAL;

	skv_proc1: WORD;

	ins_time: WORD;
	time_to_shake: TIME;

	start_stop: BLINK;
	t_r_ins: DWORD;
	t_s_ins: DWORD;
	time_r_ins: TIME;
	time_s_ins: TIME;
	shnek_up_prom: BOOL;

	prom_cleen: BOOL;

	ggg1: ggg;
	ggg2: ggg;
	ggg3: ggg;
	ggg4: ggg;
	ggg5: ggg;
	ggg6: ggg;
	ggg7: ggg;
	ggg8: ggg;
	nozzle: BOOL;
	ton1: TON;
	ton2: TON;
END_VAR
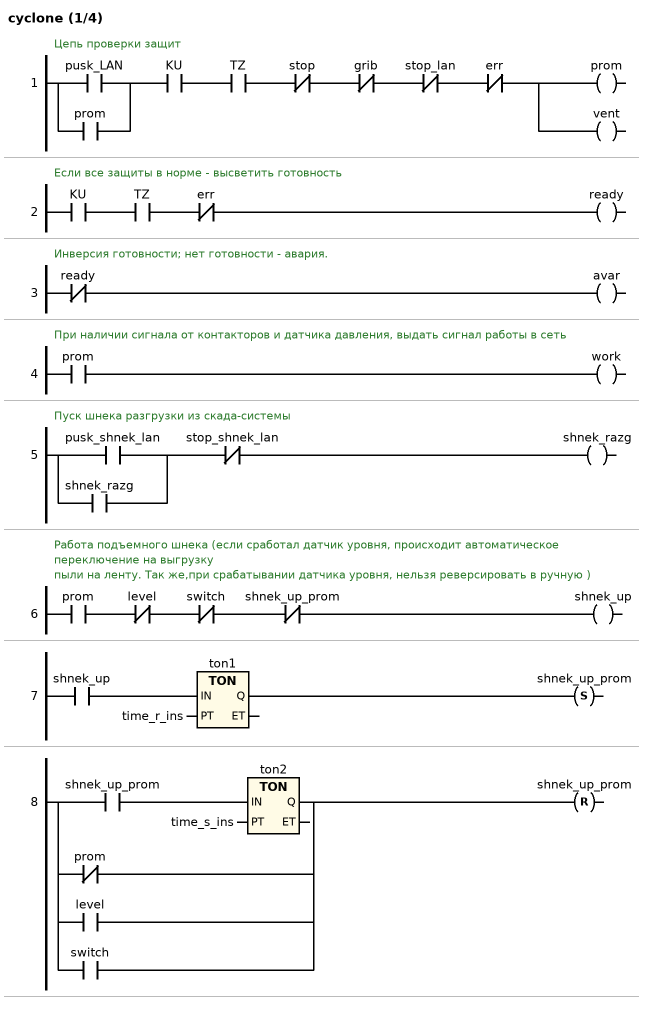
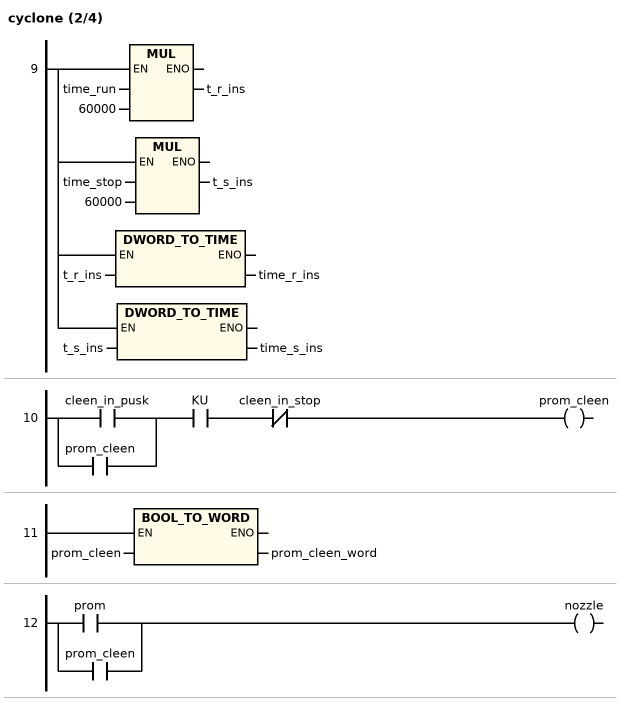
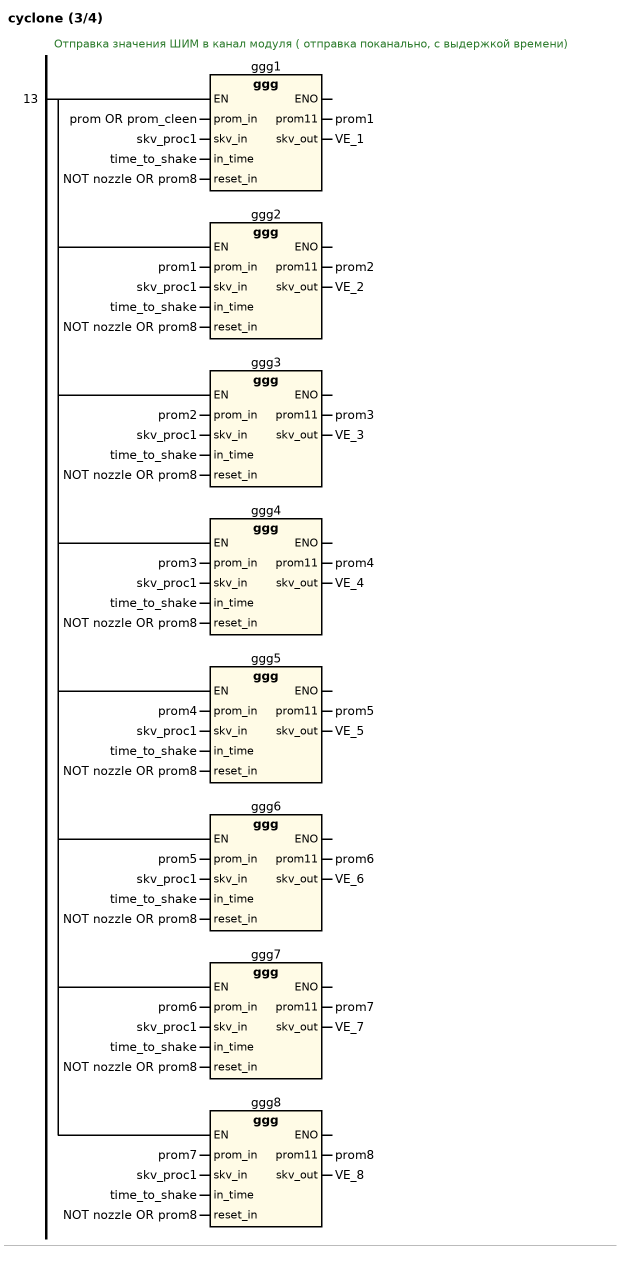
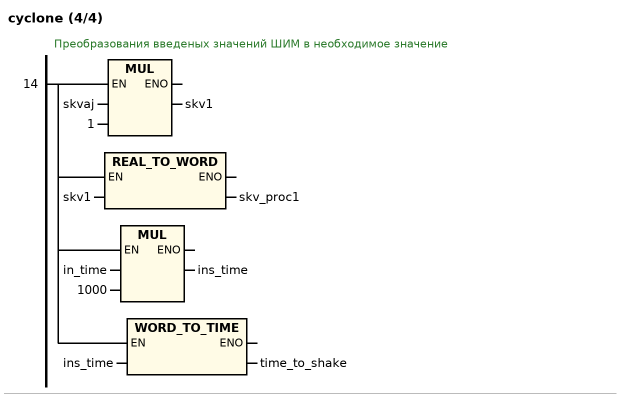
_LD_ (* Ladder Diagram *)
NETWORK 1 (* Цепь проверки защит *)
	{ [pusk_LAN] | [prom] } - [KU] - [TZ] - [/stop] - [/grib] - [/stop_lan] - [/err] --- (prom) (vent)
NETWORK 2 (* Если все защиты в норме - высветить готовность *)
	[KU] - [TZ] - [/err] --- (ready)
NETWORK 3 (* Инверсия готовности; нет готовности - авария. *)
	[/ready] --- (avar)
NETWORK 4 (* При наличии сигнала от контакторов и датчика давления, выдать сигнал работы в сеть *)
	[prom] --- (work)
NETWORK 5 (* Пуск шнека разгрузки из скада-системы *)
	{ [pusk_shnek_lan] | [shnek_razg] } - [/stop_shnek_lan] --- (shnek_razg)
NETWORK 6 (* Работа подъемного шнека (если сработал датчик уровня, происходит автоматическое переключение на выгрузку / пыли на ленту. Так же,при срабатывании датчика уровня, нельзя реверсировать в ручную ) *)
	[prom] - [/level] - [/switch] - [/shnek_up_prom] --- (shnek_up)
NETWORK 7
	[shnek_up] - ton1:TON(IN: *, PT: time_r_ins) --- (S shnek_up_prom)
NETWORK 8
	{ [shnek_up_prom] - ton2:TON(IN: *, PT: time_s_ins) | [/prom] | [level] | [switch] } --- (R shnek_up_prom)
NETWORK 9
	*
		EN --- MUL(time_run, 60000) => t_r_ins
		EN --- MUL(time_stop, 60000) => t_s_ins
		EN --- DWORD_TO_TIME(t_r_ins) => time_r_ins
		EN --- DWORD_TO_TIME(t_s_ins) => time_s_ins
NETWORK 10
	{ [cleen_in_pusk] | [prom_cleen] } - [KU] - [/cleen_in_stop] --- (prom_cleen)
NETWORK 11
	*
		EN --- BOOL_TO_WORD(prom_cleen) => prom_cleen_word
NETWORK 12
	{ [prom] | [prom_cleen] } --- (nozzle)
NETWORK 13 (* Отправка значения ШИМ в канал модуля ( отправка поканально, с выдержкой времени) *)
	*
		EN --- ggg1:ggg(prom_in: prom OR prom_cleen, skv_in: skv_proc1, in_time: time_to_shake, reset_in: NOT nozzle OR prom8, skv_out => VE_1) => prom1
		EN --- ggg2:ggg(prom_in: prom1, skv_in: skv_proc1, in_time: time_to_shake, reset_in: NOT nozzle OR prom8, skv_out => VE_2) => prom2
		EN --- ggg3:ggg(prom_in: prom2, skv_in: skv_proc1, in_time: time_to_shake, reset_in: NOT nozzle OR prom8, skv_out => VE_3) => prom3
		EN --- ggg4:ggg(prom_in: prom3, skv_in: skv_proc1, in_time: time_to_shake, reset_in: NOT nozzle OR prom8, skv_out => VE_4) => prom4
		EN --- ggg5:ggg(prom_in: prom4, skv_in: skv_proc1, in_time: time_to_shake, reset_in: NOT nozzle OR prom8, skv_out => VE_5) => prom5
		EN --- ggg6:ggg(prom_in: prom5, skv_in: skv_proc1, in_time: time_to_shake, reset_in: NOT nozzle OR prom8, skv_out => VE_6) => prom6
		EN --- ggg7:ggg(prom_in: prom6, skv_in: skv_proc1, in_time: time_to_shake, reset_in: NOT nozzle OR prom8, skv_out => VE_7) => prom7
		EN --- ggg8:ggg(prom_in: prom7, skv_in: skv_proc1, in_time: time_to_shake, reset_in: NOT nozzle OR prom8, skv_out => VE_8) => prom8
NETWORK 14 (* Преобразования введеных значений ШИМ в необходимое значение *)
	*
		EN --- MUL(skvaj, 1) => skv1
		EN --- REAL_TO_WORD(skv1) => skv_proc1
		EN --- MUL(in_time, 1000) => ins_time
		EN --- WORD_TO_TIME(ins_time) => time_to_shake
_END_LD_
(* the same logic as Structured Text *)
(* Network 1: Цепь проверки защит *)
prom := (pusk_LAN OR prom) AND KU AND TZ AND NOT stop AND NOT grib AND NOT stop_lan AND NOT err;
vent := prom;
(* Network 2: Если все защиты в норме - высветить готовность *)
ready := KU AND TZ AND NOT err;
(* Network 3: Инверсия готовности; нет готовности - авария. *)
avar := NOT ready;
(* Network 4: При наличии сигнала от контакторов и датчика давления, выдать сигнал работы в сеть *)
work := prom;
(* Network 5: Пуск шнека разгрузки из скада-системы *)
shnek_razg := (pusk_shnek_lan OR shnek_razg) AND NOT stop_shnek_lan;
(* Network 6: Работа подъемного шнека (если сработал датчик уровня, происходит автоматическое переключение на выгрузку / пыли на ленту. Так же,при срабатывании датчика уровня, нельзя реверсировать в ручную ) *)
shnek_up := prom AND NOT level AND NOT switch AND NOT shnek_up_prom;
(* Network 7 *)
ton1(IN := shnek_up, PT := time_r_ins);
IF ton1.Q THEN shnek_up_prom := TRUE; END_IF;
(* Network 8 *)
ton2(IN := shnek_up_prom, PT := time_s_ins);
IF ton2.Q OR NOT prom OR level OR switch THEN shnek_up_prom := FALSE; END_IF;
(* Network 9 *)
t_r_ins := time_run * 60000;
t_s_ins := time_stop * 60000;
time_r_ins := DWORD_TO_TIME(t_r_ins);
time_s_ins := DWORD_TO_TIME(t_s_ins);
(* Network 10 *)
prom_cleen := (cleen_in_pusk OR prom_cleen) AND KU AND NOT cleen_in_stop;
(* Network 11 *)
prom_cleen_word := BOOL_TO_WORD(prom_cleen);
(* Network 12 *)
nozzle := prom OR prom_cleen;
(* Network 13: Отправка значения ШИМ в канал модуля ( отправка поканально, с выдержкой времени) *)
ggg1(prom_in := prom OR prom_cleen, skv_in := skv_proc1, in_time := time_to_shake, reset_in := NOT nozzle OR prom8);
VE_1 := ggg1.skv_out;
prom1 := ggg1.prom11;
ggg2(prom_in := prom1, skv_in := skv_proc1, in_time := time_to_shake, reset_in := NOT nozzle OR prom8);
VE_2 := ggg2.skv_out;
prom2 := ggg2.prom11;
ggg3(prom_in := prom2, skv_in := skv_proc1, in_time := time_to_shake, reset_in := NOT nozzle OR prom8);
VE_3 := ggg3.skv_out;
prom3 := ggg3.prom11;
ggg4(prom_in := prom3, skv_in := skv_proc1, in_time := time_to_shake, reset_in := NOT nozzle OR prom8);
VE_4 := ggg4.skv_out;
prom4 := ggg4.prom11;
ggg5(prom_in := prom4, skv_in := skv_proc1, in_time := time_to_shake, reset_in := NOT nozzle OR prom8);
VE_5 := ggg5.skv_out;
prom5 := ggg5.prom11;
ggg6(prom_in := prom5, skv_in := skv_proc1, in_time := time_to_shake, reset_in := NOT nozzle OR prom8);
VE_6 := ggg6.skv_out;
prom6 := ggg6.prom11;
ggg7(prom_in := prom6, skv_in := skv_proc1, in_time := time_to_shake, reset_in := NOT nozzle OR prom8);
VE_7 := ggg7.skv_out;
prom7 := ggg7.prom11;
ggg8(prom_in := prom7, skv_in := skv_proc1, in_time := time_to_shake, reset_in := NOT nozzle OR prom8);
VE_8 := ggg8.skv_out;
prom8 := ggg8.prom11;
(* Network 14: Преобразования введеных значений ШИМ в необходимое значение *)
skv1 := skvaj * 1;
skv_proc1 := REAL_TO_WORD(skv1);
ins_time := in_time * 1000;
time_to_shake := WORD_TO_TIME(ins_time);
END_FUNCTION_BLOCK

(* POU ggg, LD *)
FUNCTION_BLOCK ggg
VAR_INPUT
	prom_in: BOOL;
	skv_in: WORD;
	in_time: TIME;
	reset_in: BOOL;
END_VAR
VAR_OUTPUT
	prom11: BOOL;
	skv_out: WORD;
END_VAR
VAR
	prom111: BOOL;
	ton11: TON;
	ton111: TON;
	rs1: RS;
END_VAR
VAR (* helpers for the ST form of the networks *)
	_p1 : BOOL;
END_VAR
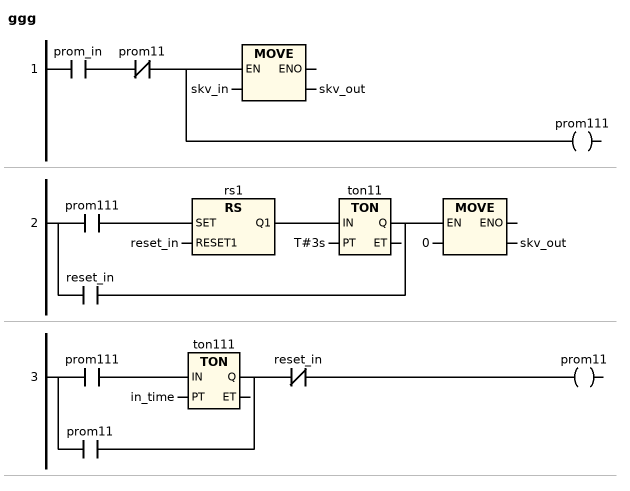
_LD_ (* Ladder Diagram *)
NETWORK 1
	[prom_in] - [/prom11] --- (prom111)
		EN --- MOVE(skv_in) => skv_out
NETWORK 2
	{ [prom111] - rs1:RS(SET: *, RESET1: reset_in) - ton11:TON(IN: *, PT: T#3s) | [reset_in] }
		EN --- MOVE(0) => skv_out
NETWORK 3
	{ [prom111] - ton111:TON(IN: *, PT: in_time) | [prom11] } - [/reset_in] --- (prom11)
_END_LD_
(* the same logic as Structured Text *)
(* Network 1 *)
_p1 := prom_in AND NOT prom11;
IF _p1 THEN
	skv_out := skv_in;
END_IF;
prom111 := _p1;
(* Network 2 *)
rs1(SET := prom111, RESET1 := reset_in);
ton11(IN := rs1.Q1, PT := T#3s);
IF ton11.Q OR reset_in THEN
	skv_out := 0;
END_IF;
(* Network 3 *)
ton111(IN := prom111, PT := in_time);
prom11 := (ton111.Q OR prom11) AND NOT reset_in;
END_FUNCTION_BLOCK

